LIN {X 0,Y 542.266,Z 432.631,A -85,B 0,C 180,E1 25597.331,E2 25597.331} C_VEL
LIN {X 0,Y 541.253,Z 430.993,A -85,B 0,C 180,E1 25597.163,E2 25597.163} C_VEL
LIN {X 0,Y 538.577,Z 428.153,A -85,B 0,C 180,E1 25596.746,E2 25596.746} C_VEL
LIN {X 0,Y 537.692,Z 425.915,A -85,B 0,C 180,E1 25596.518,E2 25596.518} C_VEL
LIN {X 0,Y 537.544,Z 425.203,A -85,B 0,C 180,E1 25596.133,E2 25596.133} C_VEL
LIN {X 0,Y 537.618,Z 425.265,A -85,B 0,C 180,E1 25592.894,E2 25592.894} C_VEL
LIN {X 0,Y 537.548,Z 425.178,A -85,B 0,C 180,E1 25589.656,E2 25589.656} C_VEL
LIN {X 0,Y 537.585,Z 425.269,A -85,B 0,C 180,E1 25586.275,E2 25586.275} C_VEL
LIN {X 0,Y 537.609,Z 425.252,A -85,B 0,C 180,E1 25582.979,E2 25582.979} C_VEL
LIN {X 0,Y 537.57,Z 425.245,A -85,B 0,C 180,E1 25579.674,E2 25579.674} C_VEL
LIN {X 0,Y 537.613,Z 425.237,A -85,B 0,C 180,E1 25576.322,E2 25576.322} C_VEL
LIN {X 0,Y 537.603,Z 425.259,A -85,B 0,C 180,E1 25573.006,E2 25573.006} C_VEL
LIN {X 0,Y 537.584,Z 425.263,A -85,B 0,C 180,E1 25569.637,E2 25569.637} C_VEL
LIN {X 0,Y 537.626,Z 425.237,A -85,B 0,C 180,E1 25566.3,E2 25566.3} C_VEL
LIN {X 0,Y 537.608,Z 425.241,A -85,B 0,C 180,E1 25562.878,E2 25562.878} C_VEL
LIN {X 0,Y 537.596,Z 425.261,A -85,B 0,C 180,E1 25559.467,E2 25559.467} C_VEL
LIN {X 0,Y 537.62,Z 425.243,A -85,B 0,C 180,E1 25556.054,E2 25556.054} C_VEL
LIN {X 0,Y 537.626,Z 425.232,A -85,B 0,C 180,E1 25552.627,E2 25552.627} C_VEL
LIN {X 0,Y 537.605,Z 425.254,A -85,B 0,C 180,E1 25549.173,E2 25549.173} C_VEL
LIN {X 0,Y 537.63,Z 425.26,A -85,B 0,C 180,E1 25545.679,E2 25545.679} C_VEL
LIN {X 0,Y 537.614,Z 425.246,A -85,B 0,C 180,E1 25542.224,E2 25542.224} C_VEL
LIN {X 0,Y 537.613,Z 425.226,A -85,B 0,C 180,E1 25538.85,E2 25538.85} C_VEL
LIN {X 0,Y 537.626,Z 425.262,A -85,B 0,C 180,E1 25535.38,E2 25535.38} C_VEL
LIN {X 0,Y 537.604,Z 425.242,A -85,B 0,C 180,E1 25531.93,E2 25531.93} C_VEL
LIN {X 0,Y 537.621,Z 425.229,A -85,B 0,C 180,E1 25528.613,E2 25528.613} C_VEL
LIN {X 0,Y 537.621,Z 425.237,A -85,B 0,C 180,E1 25525.182,E2 25525.182} C_VEL
LIN {X 0,Y 537.647,Z 425.416,A -85,B 0,C 180,E1 25522.998,E2 25522.998} C_VEL
LIN {X 0,Y 539.164,Z 429.093,A -85,B 0,C 180,E1 25522.266,E2 25522.266} C_VEL
LIN {X 0,Y 543.606,Z 438.861,A -85,B 0,C 180,E1 25520.474,E2 25520.474} C_VEL
LIN {X 0,Y 547.01,Z 446.029,A -85,B 0,C 180,E1 25519.264,E2 25519.264} C_VEL
LIN {X 0,Y 560.162,Z 465.654,A -85,B 0,C 180,E1 25517.289,E2 25517.289} C_VEL
LIN {X 0,Y 573.666,Z 487.219,A -85,B 0,C 180,E1 25515.413,E2 25515.413} C_VEL
LIN {X 0,Y 582.89,Z 503.607,A -85,B 0,C 180,E1 25514.188,E2 25514.188} C_VEL
LIN {X 0,Y 576.127,Z 736.515,A -85,B 0,C 180,E1 25510.926,E2 25510.926} C_VEL
LIN {X 0,Y 573.148,Z 839.663,A -85,B 0,C 180,E1 25509.472,E2 25509.472} C_VEL
LIN {X 0,Y 571.458,Z 865.731,A -85,B 0,C 180,E1 25508.946,E2 25508.946} C_VEL
LIN {X 0,Y 569.58,Z 887.597,A -85,B 0,C 180,E1 25508.349,E2 25508.349} C_VEL
LIN {X 0,Y 567.024,Z 912.5,A -85,B 0,C 180,E1 25507.472,E2 25507.472} C_VEL
LIN {X 0,Y 564.59,Z 933.033,A -85,B 0,C 180,E1 25506.58,E2 25506.58} C_VEL
LIN {X 0,Y 561.628,Z 955.658,A -85,B 0,C 180,E1 25505.413,E2 25505.413} C_VEL
LIN {X 0,Y 558.746,Z 975.609,A -85,B 0,C 180,E1 25504.188,E2 25504.188} C_VEL
LIN {X 0,Y 555.88,Z 994.545,A -85,B 0,C 180,E1 25502.858,E2 25502.858} C_VEL
LIN {X 0,Y 552.579,Z 1015.247,A -85,B 0,C 180,E1 25501.166,E2 25501.166} C_VEL
LIN {X 0,Y 549.796,Z 1032.714,A -85,B 0,C 180,E1 25499.529,E2 25499.529} C_VEL
LIN {X 0,Y 546.718,Z 1052.022,A -85,B 0,C 180,E1 25497.444,E2 25497.444} C_VEL
LIN {X 0,Y 544.377,Z 1067.179,A -85,B 0,C 180,E1 25495.572,E2 25495.572} C_VEL
LIN {X 0,Y 541.987,Z 1083.549,A -85,B 0,C 180,E1 25493.254,E2 25493.254} C_VEL
LIN {X 0,Y 540.268,Z 1096.427,A -85,B 0,C 180,E1 25491.155,E2 25491.155} C_VEL
LIN {X 0,Y 538.657,Z 1109.908,A -85,B 0,C 180,E1 25488.619,E2 25488.619} C_VEL
LIN {X 0,Y 537.638,Z 1119.894,A -85,B 0,C 180,E1 25486.421,E2 25486.421} C_VEL
LIN {X 0,Y 536.832,Z 1129.669,A -85,B 0,C 180,E1 25483.903,E2 25483.903} C_VEL
LIN {X 0,Y 536.342,Z 1137.217,A -85,B 0,C 180,E1 25481.506,E2 25481.506} C_VEL
LIN {X 0,Y 536.089,Z 1143.09,A -85,B 0,C 180,E1 25479.23,E2 25479.23} C_VEL
LIN {X 0,Y 535.96,Z 1148.292,A -85,B 0,C 180,E1 25476.535,E2 25476.535} C_VEL
LIN {X 0,Y 535.933,Z 1151.266,A -85,B 0,C 180,E1 25474.28,E2 25474.28} C_VEL
LIN {X 0,Y 535.914,Z 1153.221,A -85,B 0,C 180,E1 25471.711,E2 25471.711} C_VEL
LIN {X 0,Y 535.9,Z 1153.457,A -85,B 0,C 180,E1 25469.359,E2 25469.359} C_VEL
LIN {X 0,Y 535.9,Z 1152.559,A -85,B 0,C 180,E1 25467.219,E2 25467.219} C_VEL
LIN {X 0,Y 535.912,Z 1150.339,A -85,B 0,C 180,E1 25464.862,E2 25464.862} C_VEL
LIN {X 0,Y 535.975,Z 1146.441,A -85,B 0,C 180,E1 25462.389,E2 25462.389} C_VEL
LIN {X 0,Y 536.155,Z 1141.549,A -85,B 0,C 180,E1 25460.121,E2 25460.121} C_VEL
LIN {X 0,Y 536.518,Z 1134.571,A -85,B 0,C 180,E1 25457.572,E2 25457.572} C_VEL
LIN {X 0,Y 537.116,Z 1126.055,A -85,B 0,C 180,E1 25455.114,E2 25455.114} C_VEL
LIN {X 0,Y 538.018,Z 1116.198,A -85,B 0,C 180,E1 25452.701,E2 25452.701} C_VEL
LIN {X 0,Y 539.299,Z 1104.351,A -85,B 0,C 180,E1 25450.279,E2 25450.279} C_VEL
LIN {X 0,Y 540.858,Z 1091.93,A -85,B 0,C 180,E1 25448.072,E2 25448.072} C_VEL
LIN {X 0,Y 542.939,Z 1076.73,A -85,B 0,C 180,E1 25445.752,E2 25445.752} C_VEL
LIN {X 0,Y 545,Z 1062.711,A -85,B 0,C 180,E1 25443.876,E2 25443.876} C_VEL
LIN {X 0,Y 547.829,Z 1044.176,A -85,B 0,C 180,E1 25441.713,E2 25441.713} C_VEL
LIN {X 0,Y 550.405,Z 1027.597,A -85,B 0,C 180,E1 25440.028,E2 25440.028} C_VEL
LIN {X 0,Y 553.667,Z 1006.611,A -85,B 0,C 180,E1 25438.174,E2 25438.174} C_VEL
LIN {X 0,Y 556.354,Z 988.668,A -85,B 0,C 180,E1 25436.801,E2 25436.801} C_VEL
LIN {X 0,Y 559.46,Z 967.1,A -85,B 0,C 180,E1 25435.365,E2 25435.365} C_VEL
LIN {X 0,Y 562.201,Z 946.182,A -85,B 0,C 180,E1 25434.187,E2 25434.187} C_VEL
LIN {X 0,Y 564.963,Z 924.058,A -85,B 0,C 180,E1 25433.127,E2 25433.127} C_VEL
LIN {X 0,Y 567.281,Z 901.886,A -85,B 0,C 180,E1 25432.261,E2 25432.261} C_VEL
LIN {X 0,Y 569.212,Z 881.106,A -85,B 0,C 180,E1 25431.595,E2 25431.595} C_VEL
LIN {X 0,Y 571.144,Z 855.513,A -85,B 0,C 180,E1 25430.967,E2 25430.967} C_VEL
LIN {X 0,Y 572.245,Z 833.472,A -85,B 0,C 180,E1 25430.575,E2 25430.575} C_VEL
LIN {X 0,Y 578.309,Z 600.743,A -85,B 0,C 180,E1 25427.358,E2 25427.358} C_VEL
LIN {X 0,Y 580.866,Z 502.463,A -85,B 0,C 180,E1 25425.981,E2 25425.981} C_VEL
LIN {X 0,Y 566.803,Z 478.221,A -85,B 0,C 180,E1 25424.243,E2 25424.243} C_VEL
LIN {X 0,Y 553.848,Z 457.367,A -85,B 0,C 180,E1 25422.54,E2 25422.54} C_VEL
LIN {X 0,Y 546.451,Z 445.944,A -85,B 0,C 180,E1 25421.482,E2 25421.482} C_VEL
LIN {X 0,Y 540.732,Z 432.695,A -85,B 0,C 180,E1 25419.365,E2 25419.365} C_VEL
LIN {X 0,Y 537.629,Z 425.514,A -85,B 0,C 180,E1 25418.121,E2 25418.121} C_VEL
LIN {X 0,Y 537.624,Z 425.259,A -85,B 0,C 180,E1 25415.208,E2 25415.208} C_VEL
LIN {X 0,Y 537.61,Z 425.251,A -85,B 0,C 180,E1 25411.759,E2 25411.759} C_VEL
LIN {X 0,Y 537.608,Z 425.234,A -85,B 0,C 180,E1 25408.312,E2 25408.312} C_VEL
LIN {X 0,Y 537.616,Z 425.237,A -85,B 0,C 180,E1 25404.973,E2 25404.973} C_VEL
LIN {X 0,Y 537.624,Z 425.265,A -85,B 0,C 180,E1 25401.493,E2 25401.493} C_VEL
LIN {X 0,Y 537.613,Z 425.246,A -85,B 0,C 180,E1 25397.983,E2 25397.983} C_VEL
LIN {X 0,Y 537.609,Z 425.234,A -85,B 0,C 180,E1 25394.652,E2 25394.652} C_VEL
LIN {X 0,Y 537.615,Z 425.263,A -85,B 0,C 180,E1 25391.153,E2 25391.153} C_VEL
LIN {X 0,Y 537.618,Z 425.237,A -85,B 0,C 180,E1 25387.696,E2 25387.696} C_VEL
LIN {X 0,Y 537.606,Z 425.246,A -85,B 0,C 180,E1 25384.373,E2 25384.373} C_VEL
LIN {X 0,Y 537.6,Z 425.265,A -85,B 0,C 180,E1 25380.853,E2 25380.853} C_VEL
LIN {X 0,Y 537.62,Z 425.228,A -85,B 0,C 180,E1 25377.548,E2 25377.548} C_VEL
LIN {X 0,Y 537.597,Z 425.262,A -85,B 0,C 180,E1 25374.236,E2 25374.236} C_VEL
LIN {X 0,Y 537.591,Z 425.241,A -85,B 0,C 180,E1 25370.796,E2 25370.796} C_VEL
LIN {X 0,Y 537.627,Z 425.238,A -85,B 0,C 180,E1 25367.432,E2 25367.432} C_VEL
LIN {X 0,Y 537.582,Z 425.264,A -85,B 0,C 180,E1 25364.132,E2 25364.132} C_VEL
LIN {X 0,Y 537.58,Z 425.237,A -85,B 0,C 180,E1 25360.666,E2 25360.666} C_VEL
LIN {X 0,Y 537.635,Z 425.243,A -85,B 0,C 180,E1 25357.358,E2 25357.358} C_VEL
LIN {X 0,Y 537.568,Z 425.266,A -85,B 0,C 180,E1 25354.08,E2 25354.08} C_VEL
LIN {X 0,Y 537.583,Z 425.243,A -85,B 0,C 180,E1 25350.714,E2 25350.714} C_VEL
LIN {X 0,Y 537.577,Z 425.245,A -85,B 0,C 180,E1 25347.61,E2 25347.61} C_VEL
LIN {X 0,Y 537.553,Z 425.26,A -85,B 0,C 180,E1 25344.263,E2 25344.263} C_VEL
LIN {X 0,Y 537.625,Z 425.26,A -85,B 0,C 180,E1 25341.024,E2 25341.024} C_VEL
LIN {X 0,Y 537.534,Z 425.176,A -85,B 0,C 180,E1 25337.76,E2 25337.76} C_VEL
LIN {X 0,Y 537.597,Z 425.501,A -85,B 0,C 180,E1 25336.5,E2 25336.5} C_VEL
LIN {X 0,Y 538.028,Z 427.128,A -85,B 0,C 180,E1 25336.29,E2 25336.29} C_VEL
LIN {X 0,Y 540.035,Z 430.094,A -85,B 0,C 180,E1 25335.989,E2 25335.989} C_VEL
LIN {X 0,Y 541.571,Z 431.696,A -85,B 0,C 180,E1 25335.778,E2 25335.778} C_VEL
LIN {X 0,Y 544.264,Z 435.602,A -85,B 0,C 180,E1 25335.392,E2 25335.392} C_VEL
LIN {X 0,Y 546.005,Z 438.026,A -85,B 0,C 180,E1 25335.148,E2 25335.148} C_VEL
LIN {X 0,Y 556.165,Z 451.925,A -85,B 0,C 180,E1 25333.775,E2 25333.775} C_VEL
LIN {X 0,Y 568.902,Z 470.607,A -85,B 0,C 180,E1 25332.142,E2 25332.142} C_VEL
LIN {X 0,Y 578.998,Z 486.605,A -85,B 0,C 180,E1 25330.909,E2 25330.909} C_VEL
LIN {X 0,Y 581.084,Z 490.587,A -85,B 0,C 180,E1 25330.651,E2 25330.651} C_VEL
LIN {X 0,Y 574.372,Z 738.934,A -85,B 0,C 180,E1 25327.219,E2 25327.219} C_VEL
LIN {X 0,Y 573.077,Z 788.809,A -85,B 0,C 180,E1 25326.536,E2 25326.536} C_VEL
LIN {X 0,Y 572.103,Z 796.494,A -85,B 0,C 180,E1 25326.491,E2 25326.491} C_VEL
LIN {X 0,Y 566.562,Z 815.841,A -85,B 0,C 180,E1 25326.555,E2 25326.555} C_VEL
LIN {X 0,Y 565.37,Z 823.458,A -85,B 0,C 180,E1 25326.46,E2 25326.46} C_VEL
LIN {X 0,Y 563.471,Z 849.649,A -85,B 0,C 180,E1 25325.798,E2 25325.798} C_VEL
LIN {X 0,Y 561.563,Z 870.523,A -85,B 0,C 180,E1 25325.108,E2 25325.108} C_VEL
LIN {X 0,Y 558.954,Z 894.83,A -85,B 0,C 180,E1 25324.112,E2 25324.112} C_VEL
LIN {X 0,Y 556.401,Z 914.903,A -85,B 0,C 180,E1 25323.114,E2 25323.114} C_VEL
LIN {X 0,Y 553.426,Z 936.721,A -85,B 0,C 180,E1 25321.841,E2 25321.841} C_VEL
LIN {X 0,Y 550.342,Z 956.701,A -85,B 0,C 180,E1 25320.458,E2 25320.458} C_VEL
LIN {X 0,Y 547.295,Z 975.651,A -85,B 0,C 180,E1 25318.957,E2 25318.957} C_VEL
LIN {X 0,Y 544.056,Z 994.807,A -85,B 0,C 180,E1 25317.187,E2 25317.187} C_VEL
LIN {X 0,Y 541.331,Z 1010.879,A -85,B 0,C 180,E1 25315.491,E2 25315.491} C_VEL
LIN {X 0,Y 538.391,Z 1028.003,A -85,B 0,C 180,E1 25313.418,E2 25313.418} C_VEL
LIN {X 0,Y 536.15,Z 1041.437,A -85,B 0,C 180,E1 25311.555,E2 25311.555} C_VEL
LIN {X 0,Y 533.853,Z 1056.035,A -85,B 0,C 180,E1 25309.247,E2 25309.247} C_VEL
LIN {X 0,Y 532.096,Z 1067.944,A -85,B 0,C 180,E1 25307.047,E2 25307.047} C_VEL
LIN {X 0,Y 530.614,Z 1079.355,A -85,B 0,C 180,E1 25304.626,E2 25304.626} C_VEL
LIN {X 0,Y 529.486,Z 1089.213,A -85,B 0,C 180,E1 25302.1,E2 25302.1} C_VEL
LIN {X 0,Y 528.768,Z 1097.158,A -85,B 0,C 180,E1 25299.689,E2 25299.689} C_VEL
LIN {X 0,Y 528.286,Z 1104.028,A -85,B 0,C 180,E1 25297.067,E2 25297.067} C_VEL
LIN {X 0,Y 528.073,Z 1108.717,A -85,B 0,C 180,E1 25294.779,E2 25294.779} C_VEL
LIN {X 0,Y 527.969,Z 1112.732,A -85,B 0,C 180,E1 25292.062,E2 25292.062} C_VEL
LIN {X 0,Y 527.938,Z 1114.802,A -85,B 0,C 180,E1 25289.674,E2 25289.674} C_VEL
LIN {X 0,Y 527.922,Z 1115.688,A -85,B 0,C 180,E1 25287.177,E2 25287.177} C_VEL
LIN {X 0,Y 527.93,Z 1115.011,A -85,B 0,C 180,E1 25284.566,E2 25284.566} C_VEL
LIN {X 0,Y 527.961,Z 1113.176,A -85,B 0,C 180,E1 25282.272,E2 25282.272} C_VEL
LIN {X 0,Y 528.057,Z 1109.669,A -85,B 0,C 180,E1 25279.637,E2 25279.637} C_VEL
LIN {X 0,Y 528.264,Z 1104.62,A -85,B 0,C 180,E1 25277.094,E2 25277.094} C_VEL
LIN {X 0,Y 528.691,Z 1098.426,A -85,B 0,C 180,E1 25274.646,E2 25274.646} C_VEL
LIN {X 0,Y 529.407,Z 1090.185,A -85,B 0,C 180,E1 25272.07,E2 25272.07} C_VEL
LIN {X 0,Y 530.357,Z 1081.59,A -85,B 0,C 180,E1 25269.817,E2 25269.817} C_VEL
LIN {X 0,Y 531.952,Z 1069.284,A -85,B 0,C 180,E1 25267.102,E2 25267.102} C_VEL
LIN {X 0,Y 533.624,Z 1057.85,A -85,B 0,C 180,E1 25264.946,E2 25264.946} C_VEL
LIN {X 0,Y 536.117,Z 1042.465,A -85,B 0,C 180,E1 25262.449,E2 25262.449} C_VEL
LIN {X 0,Y 538.46,Z 1028.763,A -85,B 0,C 180,E1 25260.522,E2 25260.522} C_VEL
LIN {X 0,Y 541.631,Z 1010.837,A -85,B 0,C 180,E1 25258.326,E2 25258.326} C_VEL
LIN {X 0,Y 544.479,Z 994.653,A -85,B 0,C 180,E1 25256.605,E2 25256.605} C_VEL
LIN {X 0,Y 547.931,Z 975.025,A -85,B 0,C 180,E1 25254.784,E2 25254.784} C_VEL
LIN {X 0,Y 550.968,Z 956.873,A -85,B 0,C 180,E1 25253.335,E2 25253.335} C_VEL
LIN {X 0,Y 554.273,Z 936.366,A -85,B 0,C 180,E1 25251.905,E2 25251.905} C_VEL
LIN {X 0,Y 557.315,Z 914.937,A -85,B 0,C 180,E1 25250.648,E2 25250.648} C_VEL
LIN {X 0,Y 560.096,Z 894.066,A -85,B 0,C 180,E1 25249.606,E2 25249.606} C_VEL
LIN {X 0,Y 562.694,Z 870.908,A -85,B 0,C 180,E1 25248.655,E2 25248.655} C_VEL
LIN {X 0,Y 564.75,Z 849.402,A -85,B 0,C 180,E1 25247.939,E2 25247.939} C_VEL
LIN {X 0,Y 566.716,Z 823.568,A -85,B 0,C 180,E1 25247.286,E2 25247.286} C_VEL
LIN {X 0,Y 567.823,Z 801.817,A -85,B 0,C 180,E1 25246.888,E2 25246.888} C_VEL
LIN {X 0,Y 575.439,Z 551.354,A -85,B 0,C 180,E1 25243.354,E2 25243.354} C_VEL
LIN {X 0,Y 577.148,Z 493.917,A -85,B 0,C 180,E1 25242.527,E2 25242.527} C_VEL
LIN {X 0,Y 568.475,Z 480.151,A -85,B 0,C 180,E1 25241.369,E2 25241.369} C_VEL
LIN {X 0,Y 556.198,Z 462.48,A -85,B 0,C 180,E1 25239.657,E2 25239.657} C_VEL
LIN {X 0,Y 545.014,Z 447.399,A -85,B 0,C 180,E1 25237.989,E2 25237.989} C_VEL
LIN {X 0,Y 541.363,Z 442.627,A -85,B 0,C 180,E1 25237.419,E2 25237.419} C_VEL
LIN {X 0,Y 538.138,Z 438.133,A -85,B 0,C 180,E1 25236.898,E2 25236.898} C_VEL
LIN {X 0,Y 534.685,Z 434.016,A -85,B 0,C 180,E1 25236.34,E2 25236.34} C_VEL
LIN {X 0,Y 533.712,Z 432.247,A -85,B 0,C 180,E1 25236.167,E2 25236.167} C_VEL
LIN {X 0,Y 530.926,Z 429.69,A -85,B 0,C 180,E1 25235.72,E2 25235.72} C_VEL
LIN {X 0,Y 529.78,Z 427.076,A -85,B 0,C 180,E1 25235.455,E2 25235.455} C_VEL
LIN {X 0,Y 529.652,Z 426.247,A -85,B 0,C 180,E1 25235.155,E2 25235.155} C_VEL
LIN {X 0,Y 529.611,Z 426.213,A -85,B 0,C 180,E1 25231.913,E2 25231.913} C_VEL
LIN {X 0,Y 529.669,Z 426.168,A -85,B 0,C 180,E1 25228.62,E2 25228.62} C_VEL
LIN {X 0,Y 529.636,Z 426.248,A -85,B 0,C 180,E1 25225.376,E2 25225.376} C_VEL
LIN {X 0,Y 529.633,Z 426.257,A -85,B 0,C 180,E1 25221.95,E2 25221.95} C_VEL
LIN {X 0,Y 529.687,Z 426.245,A -85,B 0,C 180,E1 25218.604,E2 25218.604} C_VEL
LIN {X 0,Y 529.642,Z 426.23,A -85,B 0,C 180,E1 25215.269,E2 25215.269} C_VEL
LIN {X 0,Y 529.644,Z 426.229,A -85,B 0,C 180,E1 25211.764,E2 25211.764} C_VEL
LIN {X 0,Y 529.691,Z 426.243,A -85,B 0,C 180,E1 25208.358,E2 25208.358} C_VEL
LIN {X 0,Y 529.665,Z 426.247,A -85,B 0,C 180,E1 25204.982,E2 25204.982} C_VEL
LIN {X 0,Y 529.651,Z 426.223,A -85,B 0,C 180,E1 25201.515,E2 25201.515} C_VEL
LIN {X 0,Y 529.684,Z 426.227,A -85,B 0,C 180,E1 25198.161,E2 25198.161} C_VEL
LIN {X 0,Y 529.681,Z 426.249,A -85,B 0,C 180,E1 25194.693,E2 25194.693} C_VEL
LIN {X 0,Y 529.663,Z 426.236,A -85,B 0,C 180,E1 25191.314,E2 25191.314} C_VEL
LIN {X 0,Y 529.679,Z 426.221,A -85,B 0,C 180,E1 25187.905,E2 25187.905} C_VEL
LIN {X 0,Y 529.683,Z 426.238,A -85,B 0,C 180,E1 25184.451,E2 25184.451} C_VEL
LIN {X 0,Y 529.677,Z 426.254,A -85,B 0,C 180,E1 25180.939,E2 25180.939} C_VEL
LIN {X 0,Y 529.689,Z 426.215,A -85,B 0,C 180,E1 25177.468,E2 25177.468} C_VEL
LIN {X 0,Y 529.665,Z 426.22,A -85,B 0,C 180,E1 25174.026,E2 25174.026} C_VEL
LIN {X 0,Y 529.69,Z 426.25,A -85,B 0,C 180,E1 25170.607,E2 25170.607} C_VEL
LIN {X 0,Y 529.686,Z 426.24,A -85,B 0,C 180,E1 25167.067,E2 25167.067} C_VEL
LIN {X 0,Y 529.686,Z 426.433,A -85,B 0,C 180,E1 25164.012,E2 25164.012} C_VEL
LIN {X 0,Y 531.268,Z 430.136,A -85,B 0,C 180,E1 25163.237,E2 25163.237} C_VEL
LIN {X 0,Y 537.41,Z 443.418,A -85,B 0,C 180,E1 25160.715,E2 25160.715} C_VEL
LIN {X 0,Y 538.748,Z 446.108,A -85,B 0,C 180,E1 25160.324,E2 25160.324} C_VEL
LIN {X 0,Y 547.604,Z 458.825,A -85,B 0,C 180,E1 25158.92,E2 25158.92} C_VEL
LIN {X 0,Y 559.849,Z 477.44,A -85,B 0,C 180,E1 25157.102,E2 25157.102} C_VEL
LIN {X 0,Y 570.86,Z 495.65,A -85,B 0,C 180,E1 25155.558,E2 25155.558} C_VEL
LIN {X 0,Y 577.15,Z 506.92,A -85,B 0,C 180,E1 25154.706,E2 25154.706} C_VEL
LIN {X 0,Y 570.13,Z 737.84,A -85,B 0,C 180,E1 25151.445,E2 25151.445} C_VEL
LIN {X 0,Y 567.06,Z 839.446,A -85,B 0,C 180,E1 25149.999,E2 25149.999} C_VEL
LIN {X 0,Y 565.316,Z 865.417,A -85,B 0,C 180,E1 25149.472,E2 25149.472} C_VEL
LIN {X 0,Y 563.366,Z 887.233,A -85,B 0,C 180,E1 25148.873,E2 25148.873} C_VEL
LIN {X 0,Y 560.635,Z 912.63,A -85,B 0,C 180,E1 25147.972,E2 25147.972} C_VEL
LIN {X 0,Y 558.106,Z 933.07,A -85,B 0,C 180,E1 25147.076,E2 25147.076} C_VEL
LIN {X 0,Y 554.879,Z 956.488,A -85,B 0,C 180,E1 25145.849,E2 25145.849} C_VEL
LIN {X 0,Y 552.005,Z 975.542,A -85,B 0,C 180,E1 25144.665,E2 25144.665} C_VEL
LIN {X 0,Y 548.867,Z 995.372,A -85,B 0,C 180,E1 25143.254,E2 25143.254} C_VEL
LIN {X 0,Y 545.439,Z 1015.723,A -85,B 0,C 180,E1 25141.559,E2 25141.559} C_VEL
LIN {X 0,Y 542.351,Z 1034.232,A -85,B 0,C 180,E1 25139.792,E2 25139.792} C_VEL
LIN {X 0,Y 539.365,Z 1051.939,A -85,B 0,C 180,E1 25137.837,E2 25137.837} C_VEL
LIN {X 0,Y 536.902,Z 1066.971,A -85,B 0,C 180,E1 25135.954,E2 25135.954} C_VEL
LIN {X 0,Y 534.381,Z 1083.314,A -85,B 0,C 180,E1 25133.605,E2 25133.605} C_VEL
LIN {X 0,Y 532.543,Z 1096.174,A -85,B 0,C 180,E1 25131.477,E2 25131.477} C_VEL
LIN {X 0,Y 530.83,Z 1109.631,A -85,B 0,C 180,E1 25128.904,E2 25128.904} C_VEL
LIN {X 0,Y 529.75,Z 1119.601,A -85,B 0,C 180,E1 25126.672,E2 25126.672} C_VEL
LIN {X 0,Y 528.885,Z 1129.419,A -85,B 0,C 180,E1 25124.102,E2 25124.102} C_VEL
LIN {X 0,Y 528.372,Z 1136.924,A -85,B 0,C 180,E1 25121.682,E2 25121.682} C_VEL
LIN {X 0,Y 528.106,Z 1142.8,A -85,B 0,C 180,E1 25119.371,E2 25119.371} C_VEL
LIN {X 0,Y 527.965,Z 1148.004,A -85,B 0,C 180,E1 25116.634,E2 25116.634} C_VEL
LIN {X 0,Y 527.935,Z 1150.979,A -85,B 0,C 180,E1 25114.345,E2 25114.345} C_VEL
LIN {X 0,Y 527.922,Z 1152.896,A -85,B 0,C 180,E1 25111.845,E2 25111.845} C_VEL
LIN {X 0,Y 527.905,Z 1153.172,A -85,B 0,C 180,E1 25109.349,E2 25109.349} C_VEL
LIN {X 0,Y 527.903,Z 1152.275,A -85,B 0,C 180,E1 25107.177,E2 25107.177} C_VEL
LIN {X 0,Y 527.914,Z 1150.054,A -85,B 0,C 180,E1 25104.784,E2 25104.784} C_VEL
LIN {X 0,Y 527.992,Z 1145.945,A -85,B 0,C 180,E1 25102.163,E2 25102.163} C_VEL
LIN {X 0,Y 528.175,Z 1141.033,A -85,B 0,C 180,E1 25099.873,E2 25099.873} C_VEL
LIN {X 0,Y 528.588,Z 1133.736,A -85,B 0,C 180,E1 25097.213,E2 25097.213} C_VEL
LIN {X 0,Y 529.194,Z 1125.766,A -85,B 0,C 180,E1 25094.886,E2 25094.886} C_VEL
LIN {X 0,Y 530.1,Z 1116.369,A -85,B 0,C 180,E1 25092.548,E2 25092.548} C_VEL
LIN {X 0,Y 531.442,Z 1104.615,A -85,B 0,C 180,E1 25090.09,E2 25090.09} C_VEL
LIN {X 0,Y 532.979,Z 1092.886,A -85,B 0,C 180,E1 25087.963,E2 25087.963} C_VEL
LIN {X 0,Y 535.249,Z 1077.15,A -85,B 0,C 180,E1 25085.499,E2 25085.499} C_VEL
LIN {X 0,Y 537.402,Z 1063.189,A -85,B 0,C 180,E1 25083.597,E2 25083.597} C_VEL
LIN {X 0,Y 540.332,Z 1044.933,A -85,B 0,C 180,E1 25081.422,E2 25081.422} C_VEL
LIN {X 0,Y 543.038,Z 1028.296,A -85,B 0,C 180,E1 25079.701,E2 25079.701} C_VEL
LIN {X 0,Y 546.23,Z 1008.857,A -85,B 0,C 180,E1 25077.937,E2 25077.937} C_VEL
LIN {X 0,Y 549.187,Z 989.911,A -85,B 0,C 180,E1 25076.456,E2 25076.456} C_VEL
LIN {X 0,Y 552.38,Z 968.924,A -85,B 0,C 180,E1 25075.023,E2 25075.023} C_VEL
LIN {X 0,Y 555.395,Z 946.898,A -85,B 0,C 180,E1 25073.76,E2 25073.76} C_VEL
LIN {X 0,Y 558.219,Z 925.153,A -85,B 0,C 180,E1 25072.702,E2 25072.702} C_VEL
LIN {X 0,Y 560.785,Z 901.912,A -85,B 0,C 180,E1 25071.778,E2 25071.778} C_VEL
LIN {X 0,Y 562.747,Z 881.616,A -85,B 0,C 180,E1 25071.121,E2 25071.121} C_VEL
LIN {X 0,Y 564.78,Z 856,A -85,B 0,C 180,E1 25070.481,E2 25070.481} C_VEL
LIN {X 0,Y 565.948,Z 833.625,A -85,B 0,C 180,E1 25070.077,E2 25070.077} C_VEL
LIN {X 0,Y 572.285,Z 601.478,A -85,B 0,C 180,E1 25066.839,E2 25066.839} C_VEL
LIN {X 0,Y 574.899,Z 505.729,A -85,B 0,C 180,E1 25065.487,E2 25065.487} C_VEL
LIN {X 0,Y 560.515,Z 480.862,A -85,B 0,C 180,E1 25063.659,E2 25063.659} C_VEL
LIN {X 0,Y 548.607,Z 461.767,A -85,B 0,C 180,E1 25062.052,E2 25062.052} C_VEL
LIN {X 0,Y 538.073,Z 445.468,A -85,B 0,C 180,E1 25060.502,E2 25060.502} C_VEL
LIN {X 0,Y 532.475,Z 433.182,A -85,B 0,C 180,E1 25058.43,E2 25058.43} C_VEL
LIN {X 0,Y 529.704,Z 426.379,A -85,B 0,C 180,E1 25057.205,E2 25057.205} C_VEL
LIN {X 0,Y 529.672,Z 426.232,A -85,B 0,C 180,E1 25053.711,E2 25053.711} C_VEL
LIN {X 0,Y 529.664,Z 426.246,A -85,B 0,C 180,E1 25050.268,E2 25050.268} C_VEL
LIN {X 0,Y 529.682,Z 426.248,A -85,B 0,C 180,E1 25046.94,E2 25046.94} C_VEL
LIN {X 0,Y 529.681,Z 426.22,A -85,B 0,C 180,E1 25043.446,E2 25043.446} C_VEL
LIN {X 0,Y 529.673,Z 426.231,A -85,B 0,C 180,E1 25040.095,E2 25040.095} C_VEL
LIN {X 0,Y 529.677,Z 426.251,A -85,B 0,C 180,E1 25036.675,E2 25036.675} C_VEL
LIN {X 0,Y 529.678,Z 426.224,A -85,B 0,C 180,E1 25033.204,E2 25033.204} C_VEL
LIN {X 0,Y 529.677,Z 426.228,A -85,B 0,C 180,E1 25029.782,E2 25029.782} C_VEL
LIN {X 0,Y 529.673,Z 426.25,A -85,B 0,C 180,E1 25026.395,E2 25026.395} C_VEL
LIN {X 0,Y 529.66,Z 426.219,A -85,B 0,C 180,E1 25022.922,E2 25022.922} C_VEL
LIN {X 0,Y 529.686,Z 426.246,A -85,B 0,C 180,E1 25019.567,E2 25019.567} C_VEL
LIN {X 0,Y 529.668,Z 426.236,A -85,B 0,C 180,E1 25016.103,E2 25016.103} C_VEL
LIN {X 0,Y 529.649,Z 426.226,A -85,B 0,C 180,E1 25012.733,E2 25012.733} C_VEL
LIN {X 0,Y 529.686,Z 426.25,A -85,B 0,C 180,E1 25009.339,E2 25009.339} C_VEL
LIN {X 0,Y 529.65,Z 426.219,A -85,B 0,C 180,E1 25006.013,E2 25006.013} C_VEL
LIN {X 0,Y 529.64,Z 426.244,A -85,B 0,C 180,E1 25002.532,E2 25002.532} C_VEL
LIN {X 0,Y 529.683,Z 426.244,A -85,B 0,C 180,E1 24999.135,E2 24999.135} C_VEL
LIN {X 0,Y 529.635,Z 426.221,A -85,B 0,C 180,E1 24995.934,E2 24995.934} C_VEL
LIN {X 0,Y 529.628,Z 426.24,A -85,B 0,C 180,E1 24992.449,E2 24992.449} C_VEL
LIN {X 0,Y 529.69,Z 426.252,A -85,B 0,C 180,E1 24989.194,E2 24989.194} C_VEL
LIN {X 0,Y 529.618,Z 426.247,A -85,B 0,C 180,E1 24985.894,E2 24985.894} C_VEL
LIN {X 0,Y 529.62,Z 426.24,A -85,B 0,C 180,E1 24982.424,E2 24982.424} C_VEL
LIN {X 0,Y 529.619,Z 426.187,A -85,B 0,C 180,E1 24979.499,E2 24979.499} C_VEL
LIN {X 0,Y 529.651,Z 426.441,A -85,B 0,C 180,E1 24977.48,E2 24977.48} C_VEL
LIN {X 0,Y 530.079,Z 427.976,A -85,B 0,C 180,E1 24977.247,E2 24977.247} C_VEL
LIN {X 0,Y 532.154,Z 431.046,A -85,B 0,C 180,E1 24976.921,E2 24976.921} C_VEL
LIN {X 0,Y 533.66,Z 432.622,A -85,B 0,C 180,E1 24976.705,E2 24976.705} C_VEL
LIN {X 0,Y 536.294,Z 436.535,A -85,B 0,C 180,E1 24976.308,E2 24976.308} C_VEL
LIN {X 0,Y 537.945,Z 438.597,A -85,B 0,C 180,E1 24976.071,E2 24976.071} C_VEL
LIN {X 0,Y 551.932,Z 457.837,A -85,B 0,C 180,E1 24974.122,E2 24974.122} C_VEL
LIN {X 0,Y 564.97,Z 477.126,A -85,B 0,C 180,E1 24972.419,E2 24972.419} C_VEL
LIN {X 0,Y 574.835,Z 493.001,A -85,B 0,C 180,E1 24971.19,E2 24971.19} C_VEL
LIN {X 0,Y 575.112,Z 494.334,A -85,B 0,C 180,E1 24971.142,E2 24971.142} C_VEL
LIN {X 0,Y 568.126,Z 741.643,A -85,B 0,C 180,E1 24967.695,E2 24967.695} C_VEL
LIN {X 0,Y 566.121,Z 809.613,A -85,B 0,C 180,E1 24966.729,E2 24966.729} C_VEL
LIN {X 0,Y 565.37,Z 823.458,A -85,B 0,C 180,E1 24966.46,E2 24966.46} C_VEL
LIN {X 0,Y 563.494,Z 833.207,A -85,B 0,C 180,E1 24966.343,E2 24966.343} C_VEL
LIN {X 0,Y 558.145,Z 849.089,A -85,B 0,C 180,E1 24966.253,E2 24966.253} C_VEL
LIN {X 0,Y 556.611,Z 856.534,A -85,B 0,C 180,E1 24966.097,E2 24966.097} C_VEL
LIN {X 0,Y 556.509,Z 857.594,A -85,B 0,C 180,E1 24966.065,E2 24966.065} C_VEL
LIN {X 0,Y 554.074,Z 881.465,A -85,B 0,C 180,E1 24965.192,E2 24965.192} C_VEL
LIN {X 0,Y 551.685,Z 901.28,A -85,B 0,C 180,E1 24964.31,E2 24964.31} C_VEL
LIN {X 0,Y 548.708,Z 923.455,A -85,B 0,C 180,E1 24963.14,E2 24963.14} C_VEL
LIN {X 0,Y 545.615,Z 943.821,A -85,B 0,C 180,E1 24961.856,E2 24961.856} C_VEL
LIN {X 0,Y 542.281,Z 964.56,A -85,B 0,C 180,E1 24960.346,E2 24960.346} C_VEL
LIN {X 0,Y 538.995,Z 983.557,A -85,B 0,C 180,E1 24958.716,E2 24958.716} C_VEL
LIN {X 0,Y 535.861,Z 1001.494,A -85,B 0,C 180,E1 24956.964,E2 24956.964} C_VEL
LIN {X 0,Y 532.679,Z 1018.929,A -85,B 0,C 180,E1 24954.983,E2 24954.983} C_VEL
LIN {X 0,Y 530.113,Z 1033.496,A -85,B 0,C 180,E1 24953.099,E2 24953.099} C_VEL
LIN {X 0,Y 527.412,Z 1049.151,A -85,B 0,C 180,E1 24950.764,E2 24950.764} C_VEL
LIN {X 0,Y 525.509,Z 1060.858,A -85,B 0,C 180,E1 24948.757,E2 24948.757} C_VEL
LIN {X 0,Y 523.584,Z 1073.823,A -85,B 0,C 180,E1 24946.19,E2 24946.19} C_VEL
LIN {X 0,Y 522.325,Z 1083.463,A -85,B 0,C 180,E1 24943.937,E2 24943.937} C_VEL
LIN {X 0,Y 521.311,Z 1092.783,A -85,B 0,C 180,E1 24941.394,E2 24941.394} C_VEL
LIN {X 0,Y 520.621,Z 1100.307,A -85,B 0,C 180,E1 24938.838,E2 24938.838} C_VEL
LIN {X 0,Y 520.239,Z 1106.148,A -85,B 0,C 180,E1 24936.4,E2 24936.4} C_VEL
LIN {X 0,Y 520.009,Z 1110.997,A -85,B 0,C 180,E1 24933.664,E2 24933.664} C_VEL
LIN {X 0,Y 519.948,Z 1113.727,A -85,B 0,C 180,E1 24931.433,E2 24931.433} C_VEL
LIN {X 0,Y 519.918,Z 1115.583,A -85,B 0,C 180,E1 24928.898,E2 24928.898} C_VEL
LIN {X 0,Y 519.92,Z 1115.877,A -85,B 0,C 180,E1 24926.251,E2 24926.251} C_VEL
LIN {X 0,Y 519.947,Z 1114.936,A -85,B 0,C 180,E1 24923.929,E2 24923.929} C_VEL
LIN {X 0,Y 519.999,Z 1112.289,A -85,B 0,C 180,E1 24921.151,E2 24921.151} C_VEL
LIN {X 0,Y 520.126,Z 1108.446,A -85,B 0,C 180,E1 24918.692,E2 24918.692} C_VEL
LIN {X 0,Y 520.436,Z 1103.047,A -85,B 0,C 180,E1 24916.104,E2 24916.104} C_VEL
LIN {X 0,Y 520.997,Z 1095.872,A -85,B 0,C 180,E1 24913.498,E2 24913.498} C_VEL
LIN {X 0,Y 521.778,Z 1088.256,A -85,B 0,C 180,E1 24911.203,E2 24911.203} C_VEL
LIN {X 0,Y 523.145,Z 1077.354,A -85,B 0,C 180,E1 24908.471,E2 24908.471} C_VEL
LIN {X 0,Y 524.62,Z 1067.1,A -85,B 0,C 180,E1 24906.287,E2 24906.287} C_VEL
LIN {X 0,Y 526.881,Z 1053.31,A -85,B 0,C 180,E1 24903.757,E2 24903.757} C_VEL
LIN {X 0,Y 529.139,Z 1040.206,A -85,B 0,C 180,E1 24901.686,E2 24901.686} C_VEL
LIN {X 0,Y 532.118,Z 1024.029,A -85,B 0,C 180,E1 24899.45,E2 24899.45} C_VEL
LIN {X 0,Y 535.109,Z 1007.712,A -85,B 0,C 180,E1 24897.506,E2 24897.506} C_VEL
LIN {X 0,Y 538.498,Z 989.81,A -85,B 0,C 180,E1 24895.634,E2 24895.634} C_VEL
LIN {X 0,Y 541.882,Z 970.902,A -85,B 0,C 180,E1 24893.94,E2 24893.94} C_VEL
LIN {X 0,Y 545.258,Z 951.625,A -85,B 0,C 180,E1 24892.429,E2 24892.429} C_VEL
LIN {X 0,Y 548.595,Z 930.715,A -85,B 0,C 180,E1 24891.037,E2 24891.037} C_VEL
LIN {X 0,Y 551.606,Z 910.443,A -85,B 0,C 180,E1 24889.878,E2 24889.878} C_VEL
LIN {X 0,Y 554.66,Z 887.442,A -85,B 0,C 180,E1 24888.784,E2 24888.784} C_VEL
LIN {X 0,Y 556.918,Z 867.452,A -85,B 0,C 180,E1 24887.995,E2 24887.995} C_VEL
LIN {X 0,Y 559.256,Z 843.26,A -85,B 0,C 180,E1 24887.225,E2 24887.225} C_VEL
LIN {X 0,Y 560.842,Z 821.279,A -85,B 0,C 180,E1 24886.698,E2 24886.698} C_VEL
LIN {X 0,Y 562.007,Z 798.053,A -85,B 0,C 180,E1 24886.286,E2 24886.286} C_VEL
LIN {X 0,Y 569.944,Z 546.909,A -85,B 0,C 180,E1 24882.72,E2 24882.72} C_VEL
LIN {X 0,Y 571.44,Z 497.364,A -85,B 0,C 180,E1 24881.996,E2 24881.996} C_VEL
LIN {X 0,Y 563.163,Z 484.358,A -85,B 0,C 180,E1 24880.865,E2 24880.865} C_VEL
LIN {X 0,Y 551.891,Z 468.093,A -85,B 0,C 180,E1 24879.254,E2 24879.254} C_VEL
LIN {X 0,Y 541.102,Z 453.443,A -85,B 0,C 180,E1 24877.609,E2 24877.609} C_VEL
LIN {X 0,Y 537.066,Z 448.255,A -85,B 0,C 180,E1 24876.967,E2 24876.967} C_VEL
LIN {X 0,Y 533.515,Z 443.51,A -85,B 0,C 180,E1 24876.383,E2 24876.383} C_VEL
LIN {X 0,Y 529.862,Z 438.692,A -85,B 0,C 180,E1 24875.766,E2 24875.766} C_VEL
LIN {X 0,Y 526.909,Z 435.251,A -85,B 0,C 180,E1 24875.265,E2 24875.265} C_VEL
LIN {X 0,Y 525.771,Z 433.204,A -85,B 0,C 180,E1 24875.053,E2 24875.053} C_VEL
LIN {X 0,Y 522.929,Z 430.546,A -85,B 0,C 180,E1 24874.57,E2 24874.57} C_VEL
LIN {X 0,Y 521.822,Z 427.993,A -85,B 0,C 180,E1 24874.288,E2 24874.288} C_VEL
LIN {X 0,Y 521.673,Z 427.238,A -85,B 0,C 180,E1 24873.901,E2 24873.901} C_VEL
LIN {X 0,Y 521.72,Z 427.152,A -85,B 0,C 180,E1 24870.624,E2 24870.624} C_VEL
LIN {X 0,Y 521.69,Z 427.199,A -85,B 0,C 180,E1 24867.387,E2 24867.387} C_VEL
LIN {X 0,Y 521.689,Z 427.222,A -85,B 0,C 180,E1 24863.902,E2 24863.902} C_VEL
LIN {X 0,Y 521.748,Z 427.215,A -85,B 0,C 180,E1 24860.648,E2 24860.648} C_VEL
LIN {X 0,Y 521.706,Z 427.235,A -85,B 0,C 180,E1 24857.282,E2 24857.282} C_VEL
LIN {X 0,Y 521.705,Z 427.244,A -85,B 0,C 180,E1 24853.748,E2 24853.748} C_VEL
LIN {X 0,Y 521.746,Z 427.221,A -85,B 0,C 180,E1 24850.378,E2 24850.378} C_VEL
LIN {X 0,Y 521.727,Z 427.213,A -85,B 0,C 180,E1 24846.935,E2 24846.935} C_VEL
LIN {X 0,Y 521.713,Z 427.234,A -85,B 0,C 180,E1 24843.516,E2 24843.516} C_VEL
LIN {X 0,Y 521.75,Z 427.235,A -85,B 0,C 180,E1 24840,E2 24840} C_VEL
LIN {X 0,Y 521.74,Z 427.211,A -85,B 0,C 180,E1 24836.484,E2 24836.484} C_VEL
LIN {X 0,Y 521.724,Z 427.214,A -85,B 0,C 180,E1 24833.065,E2 24833.065} C_VEL
LIN {X 0,Y 521.735,Z 427.238,A -85,B 0,C 180,E1 24829.51,E2 24829.51} C_VEL
LIN {X 0,Y 521.738,Z 427.237,A -85,B 0,C 180,E1 24826.026,E2 24826.026} C_VEL
LIN {X 0,Y 521.739,Z 427.216,A -85,B 0,C 180,E1 24822.604,E2 24822.604} C_VEL
LIN {X 0,Y 521.734,Z 427.204,A -85,B 0,C 180,E1 24819.117,E2 24819.117} C_VEL
LIN {X 0,Y 521.735,Z 427.242,A -85,B 0,C 180,E1 24815.787,E2 24815.787} C_VEL
LIN {X 0,Y 521.731,Z 427.209,A -85,B 0,C 180,E1 24812.244,E2 24812.244} C_VEL
LIN {X 0,Y 521.741,Z 427.204,A -85,B 0,C 180,E1 24808.839,E2 24808.839} C_VEL
LIN {X 0,Y 521.731,Z 427.217,A -85,B 0,C 180,E1 24805.439,E2 24805.439} C_VEL
LIN {X 0,Y 521.823,Z 427.717,A -85,B 0,C 180,E1 24804.996,E2 24804.996} C_VEL
LIN {X 0,Y 523.457,Z 431.301,A -85,B 0,C 180,E1 24804.231,E2 24804.231} C_VEL
LIN {X 0,Y 527.948,Z 441.033,A -85,B 0,C 180,E1 24802.285,E2 24802.285} C_VEL
LIN {X 0,Y 529.954,Z 445.038,A -85,B 0,C 180,E1 24801.561,E2 24801.561} C_VEL
LIN {X 0,Y 540.872,Z 460.812,A -85,B 0,C 180,E1 24799.734,E2 24799.734} C_VEL
LIN {X 0,Y 551.915,Z 477.325,A -85,B 0,C 180,E1 24798.03,E2 24798.03} C_VEL
LIN {X 0,Y 565.109,Z 498.779,A -85,B 0,C 180,E1 24796.12,E2 24796.12} C_VEL
LIN {X 0,Y 571.456,Z 510.293,A -85,B 0,C 180,E1 24795.234,E2 24795.234} C_VEL
LIN {X 0,Y 564.184,Z 739.202,A -85,B 0,C 180,E1 24791.974,E2 24791.974} C_VEL
LIN {X 0,Y 561.026,Z 839.149,A -85,B 0,C 180,E1 24790.539,E2 24790.539} C_VEL
LIN {X 0,Y 559.226,Z 865.119,A -85,B 0,C 180,E1 24790.008,E2 24790.008} C_VEL
LIN {X 0,Y 557.22,Z 886.749,A -85,B 0,C 180,E1 24789.412,E2 24789.412} C_VEL
LIN {X 0,Y 554.443,Z 911.605,A -85,B 0,C 180,E1 24788.531,E2 24788.531} C_VEL
LIN {X 0,Y 551.817,Z 931.99,A -85,B 0,C 180,E1 24787.636,E2 24787.636} C_VEL
LIN {X 0,Y 548.583,Z 954.661,A -85,B 0,C 180,E1 24786.455,E2 24786.455} C_VEL
LIN {X 0,Y 545.454,Z 974.539,A -85,B 0,C 180,E1 24785.217,E2 24785.217} C_VEL
LIN {X 0,Y 542.266,Z 993.815,A -85,B 0,C 180,E1 24783.839,E2 24783.839} C_VEL
LIN {X 0,Y 538.663,Z 1014.374,A -85,B 0,C 180,E1 24782.128,E2 24782.128} C_VEL
LIN {X 0,Y 535.659,Z 1031.292,A -85,B 0,C 180,E1 24780.513,E2 24780.513} C_VEL
LIN {X 0,Y 532.244,Z 1050.719,A -85,B 0,C 180,E1 24778.379,E2 24778.379} C_VEL
LIN {X 0,Y 529.597,Z 1065.921,A -85,B 0,C 180,E1 24776.46,E2 24776.46} C_VEL
LIN {X 0,Y 526.91,Z 1082.383,A -85,B 0,C 180,E1 24774.079,E2 24774.079} C_VEL
LIN {X 0,Y 524.929,Z 1095.295,A -85,B 0,C 180,E1 24771.922,E2 24771.922} C_VEL
LIN {X 0,Y 523.163,Z 1108.327,A -85,B 0,C 180,E1 24769.424,E2 24769.424} C_VEL
LIN {X 0,Y 521.923,Z 1118.864,A -85,B 0,C 180,E1 24767.045,E2 24767.045} C_VEL
LIN {X 0,Y 520.989,Z 1128.726,A -85,B 0,C 180,E1 24764.448,E2 24764.448} C_VEL
LIN {X 0,Y 520.429,Z 1136.323,A -85,B 0,C 180,E1 24761.976,E2 24761.976} C_VEL
LIN {X 0,Y 520.136,Z 1142.249,A -85,B 0,C 180,E1 24759.628,E2 24759.628} C_VEL
LIN {X 0,Y 519.975,Z 1147.552,A -85,B 0,C 180,E1 24756.847,E2 24756.847} C_VEL
LIN {X 0,Y 519.937,Z 1150.576,A -85,B 0,C 180,E1 24754.522,E2 24754.522} C_VEL
LIN {X 0,Y 519.932,Z 1152.473,A -85,B 0,C 180,E1 24752.094,E2 24752.094} C_VEL
LIN {X 0,Y 519.912,Z 1152.911,A -85,B 0,C 180,E1 24749.449,E2 24749.449} C_VEL
LIN {X 0,Y 519.909,Z 1152.06,A -85,B 0,C 180,E1 24747.244,E2 24747.244} C_VEL
LIN {X 0,Y 519.918,Z 1150.003,A -85,B 0,C 180,E1 24744.925,E2 24744.925} C_VEL
LIN {X 0,Y 519.984,Z 1146.082,A -85,B 0,C 180,E1 24742.264,E2 24742.264} C_VEL
LIN {X 0,Y 520.17,Z 1141.236,A -85,B 0,C 180,E1 24739.926,E2 24739.926} C_VEL
LIN {X 0,Y 520.54,Z 1134.804,A -85,B 0,C 180,E1 24737.464,E2 24737.464} C_VEL
LIN {X 0,Y 521.203,Z 1126.292,A -85,B 0,C 180,E1 24734.876,E2 24734.876} C_VEL
LIN {X 0,Y 522.078,Z 1117.458,A -85,B 0,C 180,E1 24732.616,E2 24732.616} C_VEL
LIN {X 0,Y 523.587,Z 1104.862,A -85,B 0,C 180,E1 24729.895,E2 24729.895} C_VEL
LIN {X 0,Y 525.197,Z 1093.18,A -85,B 0,C 180,E1 24727.737,E2 24727.737} C_VEL
LIN {X 0,Y 527.452,Z 1078.342,A -85,B 0,C 180,E1 24725.351,E2 24725.351} C_VEL
LIN {X 0,Y 529.815,Z 1063.655,A -85,B 0,C 180,E1 24723.31,E2 24723.31} C_VEL
LIN {X 0,Y 532.69,Z 1046.701,A -85,B 0,C 180,E1 24721.234,E2 24721.234} C_VEL
LIN {X 0,Y 535.689,Z 1028.983,A -85,B 0,C 180,E1 24719.365,E2 24719.365} C_VEL
LIN {X 0,Y 539.012,Z 1009.735,A -85,B 0,C 180,E1 24717.581,E2 24717.581} C_VEL
LIN {X 0,Y 542.26,Z 989.725,A -85,B 0,C 180,E1 24715.996,E2 24715.996} C_VEL
LIN {X 0,Y 545.598,Z 968.702,A -85,B 0,C 180,E1 24714.547,E2 24714.547} C_VEL
LIN {X 0,Y 548.697,Z 947.055,A -85,B 0,C 180,E1 24713.293,E2 24713.293} C_VEL
LIN {X 0,Y 551.491,Z 926.339,A -85,B 0,C 180,E1 24712.272,E2 24712.272} C_VEL
LIN {X 0,Y 554.301,Z 902.185,A -85,B 0,C 180,E1 24711.293,E2 24711.293} C_VEL
LIN {X 0,Y 556.348,Z 881.837,A -85,B 0,C 180,E1 24710.627,E2 24710.627} C_VEL
LIN {X 0,Y 558.423,Z 857.011,A -85,B 0,C 180,E1 24709.994,E2 24709.994} C_VEL
LIN {X 0,Y 559.687,Z 833.948,A -85,B 0,C 180,E1 24709.571,E2 24709.571} C_VEL
LIN {X 0,Y 566.288,Z 602.803,A -85,B 0,C 180,E1 24706.317,E2 24706.317} C_VEL
LIN {X 0,Y 568.976,Z 508.989,A -85,B 0,C 180,E1 24704.983,E2 24704.983} C_VEL
LIN {X 0,Y 555.654,Z 485.882,A -85,B 0,C 180,E1 24703.248,E2 24703.248} C_VEL
LIN {X 0,Y 544.156,Z 467.292,A -85,B 0,C 180,E1 24701.661,E2 24701.661} C_VEL
LIN {X 0,Y 532.577,Z 449.793,A -85,B 0,C 180,E1 24699.966,E2 24699.966} C_VEL
LIN {X 0,Y 529.387,Z 444.828,A -85,B 0,C 180,E1 24699.42,E2 24699.42} C_VEL
LIN {X 0,Y 524.96,Z 434.873,A -85,B 0,C 180,E1 24697.692,E2 24697.692} C_VEL
LIN {X 0,Y 522.963,Z 430.569,A -85,B 0,C 180,E1 24696.896,E2 24696.896} C_VEL
LIN {X 0,Y 521.73,Z 427.326,A -85,B 0,C 180,E1 24696.238,E2 24696.238} C_VEL
LIN {X 0,Y 521.745,Z 427.212,A -85,B 0,C 180,E1 24692.844,E2 24692.844} C_VEL
LIN {X 0,Y 521.747,Z 427.211,A -85,B 0,C 180,E1 24689.381,E2 24689.381} C_VEL
LIN {X 0,Y 521.731,Z 427.236,A -85,B 0,C 180,E1 24685.91,E2 24685.91} C_VEL
LIN {X 0,Y 521.747,Z 427.229,A -85,B 0,C 180,E1 24682.419,E2 24682.419} C_VEL
LIN {X 0,Y 521.734,Z 427.21,A -85,B 0,C 180,E1 24678.898,E2 24678.898} C_VEL
LIN {X 0,Y 521.748,Z 427.222,A -85,B 0,C 180,E1 24675.428,E2 24675.428} C_VEL
LIN {X 0,Y 521.741,Z 427.236,A -85,B 0,C 180,E1 24671.945,E2 24671.945} C_VEL
LIN {X 0,Y 521.729,Z 427.204,A -85,B 0,C 180,E1 24668.486,E2 24668.486} C_VEL
LIN {X 0,Y 521.727,Z 427.231,A -85,B 0,C 180,E1 24664.947,E2 24664.947} C_VEL
LIN {X 0,Y 521.746,Z 427.226,A -85,B 0,C 180,E1 24661.428,E2 24661.428} C_VEL
LIN {X 0,Y 521.737,Z 427.207,A -85,B 0,C 180,E1 24658.023,E2 24658.023} C_VEL
LIN {X 0,Y 521.712,Z 427.243,A -85,B 0,C 180,E1 24654.611,E2 24654.611} C_VEL
LIN {X 0,Y 521.742,Z 427.205,A -85,B 0,C 180,E1 24651.292,E2 24651.292} C_VEL
LIN {X 0,Y 521.724,Z 427.23,A -85,B 0,C 180,E1 24647.942,E2 24647.942} C_VEL
LIN {X 0,Y 521.703,Z 427.236,A -85,B 0,C 180,E1 24644.549,E2 24644.549} C_VEL
LIN {X 0,Y 521.742,Z 427.206,A -85,B 0,C 180,E1 24641.214,E2 24641.214} C_VEL
LIN {X 0,Y 521.704,Z 427.242,A -85,B 0,C 180,E1 24637.935,E2 24637.935} C_VEL
LIN {X 0,Y 521.691,Z 427.235,A -85,B 0,C 180,E1 24634.453,E2 24634.453} C_VEL
LIN {X 0,Y 521.748,Z 427.21,A -85,B 0,C 180,E1 24631.122,E2 24631.122} C_VEL
LIN {X 0,Y 521.682,Z 427.227,A -85,B 0,C 180,E1 24627.905,E2 24627.905} C_VEL
LIN {X 0,Y 521.679,Z 427.237,A -85,B 0,C 180,E1 24624.358,E2 24624.358} C_VEL
LIN {X 0,Y 521.747,Z 427.238,A -85,B 0,C 180,E1 24621.054,E2 24621.054} C_VEL
LIN {X 0,Y 521.709,Z 427.394,A -85,B 0,C 180,E1 24618.509,E2 24618.509} C_VEL
LIN {X 0,Y 522.08,Z 428.9,A -85,B 0,C 180,E1 24618.258,E2 24618.258} C_VEL
LIN {X 0,Y 524.058,Z 431.94,A -85,B 0,C 180,E1 24617.929,E2 24617.929} C_VEL
LIN {X 0,Y 525.879,Z 433.69,A -85,B 0,C 180,E1 24617.657,E2 24617.657} C_VEL
LIN {X 0,Y 528.611,Z 437.643,A -85,B 0,C 180,E1 24617.229,E2 24617.229} C_VEL
LIN {X 0,Y 530.079,Z 439.527,A -85,B 0,C 180,E1 24617.007,E2 24617.007} C_VEL
LIN {X 0,Y 542.021,Z 455.841,A -85,B 0,C 180,E1 24615.262,E2 24615.262} C_VEL
LIN {X 0,Y 553.956,Z 472.819,A -85,B 0,C 180,E1 24613.63,E2 24613.63} C_VEL
LIN {X 0,Y 566.667,Z 492.542,A -85,B 0,C 180,E1 24611.983,E2 24611.983} C_VEL
LIN {X 0,Y 569.214,Z 497.09,A -85,B 0,C 180,E1 24611.656,E2 24611.656} C_VEL
LIN {X 0,Y 561.932,Z 743.819,A -85,B 0,C 180,E1 24608.189,E2 24608.189} C_VEL
LIN {X 0,Y 559.894,Z 810.012,A -85,B 0,C 180,E1 24607.239,E2 24607.239} C_VEL
LIN {X 0,Y 558.381,Z 834.747,A -85,B 0,C 180,E1 24606.714,E2 24606.714} C_VEL
LIN {X 0,Y 556.647,Z 855.872,A -85,B 0,C 180,E1 24606.119,E2 24606.119} C_VEL
LIN {X 0,Y 556.509,Z 857.594,A -85,B 0,C 180,E1 24606.065,E2 24606.065} C_VEL
LIN {X 0,Y 555.066,Z 865.043,A -85,B 0,C 180,E1 24605.882,E2 24605.882} C_VEL
LIN {X 0,Y 548.247,Z 883.715,A -85,B 0,C 180,E1 24605.552,E2 24605.552} C_VEL
LIN {X 0,Y 546.606,Z 890.898,A -85,B 0,C 180,E1 24605.314,E2 24605.314} C_VEL
LIN {X 0,Y 543.529,Z 913.618,A -85,B 0,C 180,E1 24604.195,E2 24604.195} C_VEL
LIN {X 0,Y 540.671,Z 933.058,A -85,B 0,C 180,E1 24603.063,E2 24603.063} C_VEL
LIN {X 0,Y 537.072,Z 955.221,A -85,B 0,C 180,E1 24601.544,E2 24601.544} C_VEL
LIN {X 0,Y 534.084,Z 972.41,A -85,B 0,C 180,E1 24600.177,E2 24600.177} C_VEL
LIN {X 0,Y 530.582,Z 991.792,A -85,B 0,C 180,E1 24598.414,E2 24598.414} C_VEL
LIN {X 0,Y 527.374,Z 1008.761,A -85,B 0,C 180,E1 24596.62,E2 24596.62} C_VEL
LIN {X 0,Y 524.239,Z 1025.79,A -85,B 0,C 180,E1 24594.57,E2 24594.57} C_VEL
LIN {X 0,Y 521.375,Z 1041.058,A -85,B 0,C 180,E1 24592.424,E2 24592.424} C_VEL
LIN {X 0,Y 518.934,Z 1055.116,A -85,B 0,C 180,E1 24590.176,E2 24590.176} C_VEL
LIN {X 0,Y 516.794,Z 1067.783,A -85,B 0,C 180,E1 24587.8,E2 24587.8} C_VEL
LIN {X 0,Y 515.242,Z 1078.285,A -85,B 0,C 180,E1 24585.534,E2 24585.534} C_VEL
LIN {X 0,Y 513.857,Z 1088.9,A -85,B 0,C 180,E1 24582.816,E2 24582.816} C_VEL
LIN {X 0,Y 513.073,Z 1096.283,A -85,B 0,C 180,E1 24580.556,E2 24580.556} C_VEL
LIN {X 0,Y 512.464,Z 1103.565,A -85,B 0,C 180,E1 24577.85,E2 24577.85} C_VEL
LIN {X 0,Y 512.145,Z 1108.772,A -85,B 0,C 180,E1 24575.31,E2 24575.31} C_VEL
LIN {X 0,Y 512.006,Z 1112.471,A -85,B 0,C 180,E1 24572.91,E2 24572.91} C_VEL
LIN {X 0,Y 511.971,Z 1115.161,A -85,B 0,C 180,E1 24570.112,E2 24570.112} C_VEL
LIN {X 0,Y 511.932,Z 1116.141,A -85,B 0,C 180,E1 24567.761,E2 24567.761} C_VEL
LIN {X 0,Y 511.919,Z 1115.957,A -85,B 0,C 180,E1 24565.182,E2 24565.182} C_VEL
LIN {X 0,Y 511.948,Z 1114.212,A -85,B 0,C 180,E1 24562.594,E2 24562.594} C_VEL
LIN {X 0,Y 512.016,Z 1111.57,A -85,B 0,C 180,E1 24560.332,E2 24560.332} C_VEL
LIN {X 0,Y 512.227,Z 1107.231,A -85,B 0,C 180,E1 24557.715,E2 24557.715} C_VEL
LIN {X 0,Y 512.647,Z 1101.164,A -85,B 0,C 180,E1 24555.081,E2 24555.081} C_VEL
LIN {X 0,Y 513.305,Z 1094.26,A -85,B 0,C 180,E1 24552.65,E2 24552.65} C_VEL
LIN {X 0,Y 514.468,Z 1084.439,A -85,B 0,C 180,E1 24549.84,E2 24549.84} C_VEL
LIN {X 0,Y 515.797,Z 1074.921,A -85,B 0,C 180,E1 24547.549,E2 24547.549} C_VEL
LIN {X 0,Y 517.912,Z 1061.82,A -85,B 0,C 180,E1 24544.866,E2 24544.866} C_VEL
LIN {X 0,Y 520.026,Z 1049.894,A -85,B 0,C 180,E1 24542.766,E2 24542.766} C_VEL
LIN {X 0,Y 522.877,Z 1034.745,A -85,B 0,C 180,E1 24540.438,E2 24540.438} C_VEL
LIN {X 0,Y 525.79,Z 1019.57,A -85,B 0,C 180,E1 24538.426,E2 24538.426} C_VEL
LIN {X 0,Y 529.275,Z 1002.06,A -85,B 0,C 180,E1 24536.391,E2 24536.391} C_VEL
LIN {X 0,Y 532.665,Z 984.259,A -85,B 0,C 180,E1 24534.613,E2 24534.613} C_VEL
LIN {X 0,Y 536.292,Z 965.127,A -85,B 0,C 180,E1 24532.939,E2 24532.939} C_VEL
LIN {X 0,Y 539.838,Z 944.94,A -85,B 0,C 180,E1 24531.438,E2 24531.438} C_VEL
LIN {X 0,Y 542.974,Z 925.97,A -85,B 0,C 180,E1 24530.214,E2 24530.214} C_VEL
LIN {X 0,Y 546.312,Z 903.649,A -85,B 0,C 180,E1 24528.993,E2 24528.993} C_VEL
LIN {X 0,Y 548.862,Z 884.433,A -85,B 0,C 180,E1 24528.112,E2 24528.112} C_VEL
LIN {X 0,Y 551.336,Z 863.134,A -85,B 0,C 180,E1 24527.291,E2 24527.291} C_VEL
LIN {X 0,Y 553.556,Z 839.196,A -85,B 0,C 180,E1 24526.568,E2 24526.568} C_VEL
LIN {X 0,Y 555.052,Z 818.679,A -85,B 0,C 180,E1 24526.092,E2 24526.092} C_VEL
LIN {X 0,Y 556.377,Z 789.17,A -85,B 0,C 180,E1 24525.603,E2 24525.603} C_VEL
LIN {X 0,Y 564.552,Z 541.549,A -85,B 0,C 180,E1 24522.061,E2 24522.061} C_VEL
LIN {X 0,Y 565.821,Z 500.887,A -85,B 0,C 180,E1 24521.459,E2 24521.459} C_VEL
LIN {X 0,Y 556.427,Z 486.424,A -85,B 0,C 180,E1 24520.141,E2 24520.141} C_VEL
LIN {X 0,Y 544.779,Z 469.693,A -85,B 0,C 180,E1 24518.41,E2 24518.41} C_VEL
LIN {X 0,Y 534.186,Z 455.454,A -85,B 0,C 180,E1 24516.73,E2 24516.73} C_VEL
LIN {X 0,Y 529.427,Z 449.298,A -85,B 0,C 180,E1 24515.937,E2 24515.937} C_VEL
LIN {X 0,Y 526.358,Z 445.234,A -85,B 0,C 180,E1 24515.408,E2 24515.408} C_VEL
LIN {X 0,Y 523.054,Z 441.004,A -85,B 0,C 180,E1 24514.827,E2 24514.827} C_VEL
LIN {X 0,Y 521.87,Z 439.557,A -85,B 0,C 180,E1 24514.617,E2 24514.617} C_VEL
LIN {X 0,Y 518.936,Z 436.003,A -85,B 0,C 180,E1 24514.088,E2 24514.088} C_VEL
LIN {X 0,Y 518.014,Z 434.359,A -85,B 0,C 180,E1 24513.907,E2 24513.907} C_VEL
LIN {X 0,Y 515.235,Z 431.961,A -85,B 0,C 180,E1 24513.412,E2 24513.412} C_VEL
LIN {X 0,Y 513.944,Z 429.132,A -85,B 0,C 180,E1 24513.103,E2 24513.103} C_VEL
LIN {X 0,Y 513.796,Z 428.243,A -85,B 0,C 180,E1 24512.753,E2 24512.753} C_VEL
LIN {X 0,Y 513.738,Z 428.134,A -85,B 0,C 180,E1 24509.5,E2 24509.5} C_VEL
LIN {X 0,Y 513.751,Z 428.237,A -85,B 0,C 180,E1 24505.95,E2 24505.95} C_VEL
LIN {X 0,Y 513.806,Z 428.225,A -85,B 0,C 180,E1 24502.543,E2 24502.543} C_VEL
LIN {X 0,Y 513.78,Z 428.214,A -85,B 0,C 180,E1 24499.084,E2 24499.084} C_VEL
LIN {X 0,Y 513.757,Z 428.204,A -85,B 0,C 180,E1 24495.696,E2 24495.696} C_VEL
LIN {X 0,Y 513.803,Z 428.208,A -85,B 0,C 180,E1 24492.332,E2 24492.332} C_VEL
LIN {X 0,Y 513.799,Z 428.23,A -85,B 0,C 180,E1 24488.844,E2 24488.844} C_VEL
LIN {X 0,Y 513.771,Z 428.218,A -85,B 0,C 180,E1 24485.472,E2 24485.472} C_VEL
LIN {X 0,Y 513.796,Z 428.195,A -85,B 0,C 180,E1 24482.007,E2 24482.007} C_VEL
LIN {X 0,Y 513.806,Z 428.21,A -85,B 0,C 180,E1 24478.55,E2 24478.55} C_VEL
LIN {X 0,Y 513.787,Z 428.225,A -85,B 0,C 180,E1 24475.088,E2 24475.088} C_VEL
LIN {X 0,Y 513.795,Z 428.204,A -85,B 0,C 180,E1 24471.607,E2 24471.607} C_VEL
LIN {X 0,Y 513.798,Z 428.199,A -85,B 0,C 180,E1 24468.204,E2 24468.204} C_VEL
LIN {X 0,Y 513.807,Z 428.218,A -85,B 0,C 180,E1 24464.653,E2 24464.653} C_VEL
LIN {X 0,Y 513.799,Z 428.231,A -85,B 0,C 180,E1 24461.049,E2 24461.049} C_VEL
LIN {X 0,Y 513.811,Z 428.189,A -85,B 0,C 180,E1 24457.457,E2 24457.457} C_VEL
LIN {X 0,Y 513.788,Z 428.195,A -85,B 0,C 180,E1 24454.031,E2 24454.031} C_VEL
LIN {X 0,Y 513.81,Z 428.225,A -85,B 0,C 180,E1 24450.505,E2 24450.505} C_VEL
LIN {X 0,Y 513.808,Z 428.217,A -85,B 0,C 180,E1 24446.983,E2 24446.983} C_VEL
LIN {X 0,Y 513.848,Z 428.62,A -85,B 0,C 180,E1 24446.151,E2 24446.151} C_VEL
LIN {X 0,Y 515.426,Z 432.153,A -85,B 0,C 180,E1 24445.361,E2 24445.361} C_VEL
LIN {X 0,Y 520.346,Z 442.612,A -85,B 0,C 180,E1 24443.163,E2 24443.163} C_VEL
LIN {X 0,Y 521.812,Z 445.172,A -85,B 0,C 180,E1 24442.734,E2 24442.734} C_VEL
LIN {X 0,Y 532.356,Z 459.924,A -85,B 0,C 180,E1 24440.887,E2 24440.887} C_VEL
LIN {X 0,Y 544.74,Z 478.439,A -85,B 0,C 180,E1 24438.884,E2 24438.884} C_VEL
LIN {X 0,Y 555.904,Z 496.217,A -85,B 0,C 180,E1 24437.199,E2 24437.199} C_VEL
LIN {X 0,Y 565.816,Z 513.584,A -85,B 0,C 180,E1 24435.773,E2 24435.773} C_VEL
LIN {X 0,Y 558.258,Z 741.606,A -85,B 0,C 180,E1 24432.499,E2 24432.499} C_VEL
LIN {X 0,Y 555.046,Z 838.876,A -85,B 0,C 180,E1 24431.091,E2 24431.091} C_VEL
LIN {X 0,Y 553.188,Z 864.837,A -85,B 0,C 180,E1 24430.557,E2 24430.557} C_VEL
LIN {X 0,Y 551.131,Z 886.247,A -85,B 0,C 180,E1 24429.964,E2 24429.964} C_VEL
LIN {X 0,Y 548.241,Z 911.118,A -85,B 0,C 180,E1 24429.081,E2 24429.081} C_VEL
LIN {X 0,Y 545.435,Z 932.048,A -85,B 0,C 180,E1 24428.155,E2 24428.155} C_VEL
LIN {X 0,Y 542.061,Z 954.643,A -85,B 0,C 180,E1 24426.966,E2 24426.966} C_VEL
LIN {X 0,Y 538.643,Z 975.436,A -85,B 0,C 180,E1 24425.654,E2 24425.654} C_VEL
LIN {X 0,Y 535.107,Z 995.941,A -85,B 0,C 180,E1 24424.16,E2 24424.16} C_VEL
LIN {X 0,Y 531.481,Z 1015.476,A -85,B 0,C 180,E1 24422.488,E2 24422.488} C_VEL
LIN {X 0,Y 528.163,Z 1033.388,A -85,B 0,C 180,E1 24420.74,E2 24420.74} C_VEL
LIN {X 0,Y 524.794,Z 1051.481,A -85,B 0,C 180,E1 24418.694,E2 24418.694} C_VEL
LIN {X 0,Y 522.039,Z 1066.586,A -85,B 0,C 180,E1 24416.751,E2 24416.751} C_VEL
LIN {X 0,Y 519.224,Z 1082.879,A -85,B 0,C 180,E1 24414.337,E2 24414.337} C_VEL
LIN {X 0,Y 517.156,Z 1095.712,A -85,B 0,C 180,E1 24412.149,E2 24412.149} C_VEL
LIN {X 0,Y 515.229,Z 1109.128,A -85,B 0,C 180,E1 24409.499,E2 24409.499} C_VEL
LIN {X 0,Y 514.006,Z 1119.075,A -85,B 0,C 180,E1 24407.199,E2 24407.199} C_VEL
LIN {X 0,Y 513.029,Z 1128.817,A -85,B 0,C 180,E1 24404.562,E2 24404.562} C_VEL
LIN {X 0,Y 512.444,Z 1136.354,A -85,B 0,C 180,E1 24402.051,E2 24402.051} C_VEL
LIN {X 0,Y 512.127,Z 1142.484,A -85,B 0,C 180,E1 24399.553,E2 24399.553} C_VEL
LIN {X 0,Y 511.976,Z 1147.428,A -85,B 0,C 180,E1 24396.842,E2 24396.842} C_VEL
LIN {X 0,Y 511.94,Z 1150.406,A -85,B 0,C 180,E1 24394.481,E2 24394.481} C_VEL
LIN {X 0,Y 511.932,Z 1152.325,A -85,B 0,C 180,E1 24391.903,E2 24391.903} C_VEL
LIN {X 0,Y 511.917,Z 1152.604,A -85,B 0,C 180,E1 24389.329,E2 24389.329} C_VEL
LIN {X 0,Y 511.912,Z 1151.706,A -85,B 0,C 180,E1 24387.089,E2 24387.089} C_VEL
LIN {X 0,Y 511.922,Z 1149.484,A -85,B 0,C 180,E1 24384.62,E2 24384.62} C_VEL
LIN {X 0,Y 512.013,Z 1145.372,A -85,B 0,C 180,E1 24381.917,E2 24381.917} C_VEL
LIN {X 0,Y 512.198,Z 1140.682,A -85,B 0,C 180,E1 24379.654,E2 24379.654} C_VEL
LIN {X 0,Y 512.631,Z 1133.86,A -85,B 0,C 180,E1 24377.038,E2 24377.038} C_VEL
LIN {X 0,Y 513.327,Z 1125.559,A -85,B 0,C 180,E1 24374.523,E2 24374.523} C_VEL
LIN {X 0,Y 514.332,Z 1116.189,A -85,B 0,C 180,E1 24372.112,E2 24372.112} C_VEL
LIN {X 0,Y 515.811,Z 1104.511,A -85,B 0,C 180,E1 24369.578,E2 24369.578} C_VEL
LIN {X 0,Y 517.526,Z 1092.816,A -85,B 0,C 180,E1 24367.388,E2 24367.388} C_VEL
LIN {X 0,Y 519.945,Z 1077.671,A -85,B 0,C 180,E1 24364.927,E2 24364.927} C_VEL
LIN {X 0,Y 522.435,Z 1063.025,A -85,B 0,C 180,E1 24362.87,E2 24362.87} C_VEL
LIN {X 0,Y 525.512,Z 1045.626,A -85,B 0,C 180,E1 24360.725,E2 24360.725} C_VEL
LIN {X 0,Y 528.564,Z 1028.534,A -85,B 0,C 180,E1 24358.906,E2 24358.906} C_VEL
LIN {X 0,Y 532.031,Z 1009.251,A -85,B 0,C 180,E1 24357.102,E2 24357.102} C_VEL
LIN {X 0,Y 535.35,Z 989.646,A -85,B 0,C 180,E1 24355.533,E2 24355.533} C_VEL
LIN {X 0,Y 538.769,Z 968.991,A -85,B 0,C 180,E1 24354.094,E2 24354.094} C_VEL
LIN {X 0,Y 541.996,Z 947.479,A -85,B 0,C 180,E1 24352.83,E2 24352.83} C_VEL
LIN {X 0,Y 544.726,Z 927.992,A -85,B 0,C 180,E1 24351.853,E2 24351.853} C_VEL
LIN {X 0,Y 547.75,Z 903.423,A -85,B 0,C 180,E1 24350.831,E2 24350.831} C_VEL
LIN {X 0,Y 549.918,Z 882.761,A -85,B 0,C 180,E1 24350.142,E2 24350.142} C_VEL
LIN {X 0,Y 552.064,Z 858.702,A -85,B 0,C 180,E1 24349.51,E2 24349.51} C_VEL
LIN {X 0,Y 553.464,Z 834.376,A -85,B 0,C 180,E1 24349.055,E2 24349.055} C_VEL
LIN {X 0,Y 560.347,Z 603.705,A -85,B 0,C 180,E1 24345.779,E2 24345.779} C_VEL
LIN {X 0,Y 563.104,Z 512.19,A -85,B 0,C 180,E1 24344.468,E2 24344.468} C_VEL
LIN {X 0,Y 550.368,Z 490.134,A -85,B 0,C 180,E1 24342.767,E2 24342.767} C_VEL
LIN {X 0,Y 537.748,Z 469.57,A -85,B 0,C 180,E1 24340.971,E2 24340.971} C_VEL
LIN {X 0,Y 525.68,Z 451.504,A -85,B 0,C 180,E1 24339.143,E2 24339.143} C_VEL
LIN {X 0,Y 521.11,Z 444.558,A -85,B 0,C 180,E1 24338.369,E2 24338.369} C_VEL
LIN {X 0,Y 516.561,Z 434.972,A -85,B 0,C 180,E1 24336.597,E2 24336.597} C_VEL
LIN {X 0,Y 514.895,Z 431.397,A -85,B 0,C 180,E1 24335.907,E2 24335.907} C_VEL
LIN {X 0,Y 513.829,Z 428.377,A -85,B 0,C 180,E1 24335.307,E2 24335.307} C_VEL
LIN {X 0,Y 513.79,Z 428.213,A -85,B 0,C 180,E1 24331.83,E2 24331.83} C_VEL
LIN {X 0,Y 513.796,Z 428.197,A -85,B 0,C 180,E1 24328.349,E2 24328.349} C_VEL
LIN {X 0,Y 513.801,Z 428.198,A -85,B 0,C 180,E1 24324.857,E2 24324.857} C_VEL
LIN {X 0,Y 513.809,Z 428.229,A -85,B 0,C 180,E1 24321.341,E2 24321.341} C_VEL
LIN {X 0,Y 513.796,Z 428.214,A -85,B 0,C 180,E1 24317.79,E2 24317.79} C_VEL
LIN {X 0,Y 513.809,Z 428.192,A -85,B 0,C 180,E1 24314.273,E2 24314.273} C_VEL
LIN {X 0,Y 513.791,Z 428.226,A -85,B 0,C 180,E1 24310.768,E2 24310.768} C_VEL
LIN {X 0,Y 513.806,Z 428.207,A -85,B 0,C 180,E1 24307.267,E2 24307.267} C_VEL
LIN {X 0,Y 513.801,Z 428.195,A -85,B 0,C 180,E1 24303.794,E2 24303.794} C_VEL
LIN {X 0,Y 513.787,Z 428.23,A -85,B 0,C 180,E1 24300.335,E2 24300.335} C_VEL
LIN {X 0,Y 513.776,Z 428.199,A -85,B 0,C 180,E1 24296.765,E2 24296.765} C_VEL
LIN {X 0,Y 513.813,Z 428.207,A -85,B 0,C 180,E1 24293.295,E2 24293.295} C_VEL
LIN {X 0,Y 513.799,Z 428.223,A -85,B 0,C 180,E1 24289.799,E2 24289.799} C_VEL
LIN {X 0,Y 513.76,Z 428.195,A -85,B 0,C 180,E1 24286.379,E2 24286.379} C_VEL
LIN {X 0,Y 513.784,Z 428.224,A -85,B 0,C 180,E1 24282.91,E2 24282.91} C_VEL
LIN {X 0,Y 513.804,Z 428.216,A -85,B 0,C 180,E1 24279.495,E2 24279.495} C_VEL
LIN {X 0,Y 513.749,Z 428.198,A -85,B 0,C 180,E1 24276.17,E2 24276.17} C_VEL
LIN {X 0,Y 513.775,Z 428.22,A -85,B 0,C 180,E1 24272.784,E2 24272.784} C_VEL
LIN {X 0,Y 513.781,Z 428.23,A -85,B 0,C 180,E1 24269.473,E2 24269.473} C_VEL
LIN {X 0,Y 513.737,Z 428.217,A -85,B 0,C 180,E1 24266.176,E2 24266.176} C_VEL
LIN {X 0,Y 513.782,Z 428.206,A -85,B 0,C 180,E1 24262.893,E2 24262.893} C_VEL
LIN {X 0,Y 513.742,Z 428.26,A -85,B 0,C 180,E1 24259.673,E2 24259.673} C_VEL
LIN {X 0,Y 513.937,Z 429.147,A -85,B 0,C 180,E1 24259.39,E2 24259.39} C_VEL
LIN {X 0,Y 515.773,Z 432.492,A -85,B 0,C 180,E1 24259.024,E2 24259.024} C_VEL
LIN {X 0,Y 517.945,Z 434.619,A -85,B 0,C 180,E1 24258.682,E2 24258.682} C_VEL
LIN {X 0,Y 520.459,Z 438.428,A -85,B 0,C 180,E1 24258.265,E2 24258.265} C_VEL
LIN {X 0,Y 522.42,Z 440.669,A -85,B 0,C 180,E1 24257.96,E2 24257.96} C_VEL
LIN {X 0,Y 534.176,Z 456.643,A -85,B 0,C 180,E1 24256.165,E2 24256.165} C_VEL
LIN {X 0,Y 544.649,Z 471.38,A -85,B 0,C 180,E1 24254.67,E2 24254.67} C_VEL
LIN {X 0,Y 557.855,Z 491.176,A -85,B 0,C 180,E1 24252.892,E2 24252.892} C_VEL
LIN {X 0,Y 563.341,Z 500.486,A -85,B 0,C 180,E1 24252.173,E2 24252.173} C_VEL
LIN {X 0,Y 555.773,Z 746.25,A -85,B 0,C 180,E1 24248.69,E2 24248.69} C_VEL
LIN {X 0,Y 553.707,Z 810.457,A -85,B 0,C 180,E1 24247.759,E2 24247.759} C_VEL
LIN {X 0,Y 552.14,Z 835.113,A -85,B 0,C 180,E1 24247.231,E2 24247.231} C_VEL
LIN {X 0,Y 550.328,Z 856.441,A -85,B 0,C 180,E1 24246.625,E2 24246.625} C_VEL
LIN {X 0,Y 547.798,Z 880.807,A -85,B 0,C 180,E1 24245.739,E2 24245.739} C_VEL
LIN {X 0,Y 546.606,Z 890.898,A -85,B 0,C 180,E1 24245.314,E2 24245.314} C_VEL
LIN {X 0,Y 544.934,Z 898.088,A -85,B 0,C 180,E1 24245.059,E2 24245.059} C_VEL
LIN {X 0,Y 537.586,Z 916.12,A -85,B 0,C 180,E1 24244.525,E2 24244.525} C_VEL
LIN {X 0,Y 535.739,Z 922.985,A -85,B 0,C 180,E1 24244.197,E2 24244.197} C_VEL
LIN {X 0,Y 532.362,Z 943.69,A -85,B 0,C 180,E1 24242.875,E2 24242.875} C_VEL
LIN {X 0,Y 528.991,Z 963.106,A -85,B 0,C 180,E1 24241.446,E2 24241.446} C_VEL
LIN {X 0,Y 525.259,Z 983.031,A -85,B 0,C 180,E1 24239.729,E2 24239.729} C_VEL
LIN {X 0,Y 522.018,Z 999.991,A -85,B 0,C 180,E1 24238.05,E2 24238.05} C_VEL
LIN {X 0,Y 518.439,Z 1018.233,A -85,B 0,C 180,E1 24235.964,E2 24235.964} C_VEL
LIN {X 0,Y 515.508,Z 1033.193,A -85,B 0,C 180,E1 24233.997,E2 24233.997} C_VEL
LIN {X 0,Y 512.424,Z 1049.468,A -85,B 0,C 180,E1 24231.521,E2 24231.521} C_VEL
LIN {X 0,Y 510.186,Z 1061.829,A -85,B 0,C 180,E1 24229.343,E2 24229.343} C_VEL
LIN {X 0,Y 507.974,Z 1075.228,A -85,B 0,C 180,E1 24226.584,E2 24226.584} C_VEL
LIN {X 0,Y 506.604,Z 1084.714,A -85,B 0,C 180,E1 24224.281,E2 24224.281} C_VEL
LIN {X 0,Y 505.425,Z 1094.284,A -85,B 0,C 180,E1 24221.526,E2 24221.526} C_VEL
LIN {X 0,Y 504.711,Z 1101.389,A -85,B 0,C 180,E1 24219.004,E2 24219.004} C_VEL
LIN {X 0,Y 504.253,Z 1107.605,A -85,B 0,C 180,E1 24216.261,E2 24216.261} C_VEL
LIN {X 0,Y 504.029,Z 1111.881,A -85,B 0,C 180,E1 24213.64,E2 24213.64} C_VEL
LIN {X 0,Y 503.959,Z 1114.496,A -85,B 0,C 180,E1 24211.364,E2 24211.364} C_VEL
LIN {X 0,Y 503.922,Z 1116.257,A -85,B 0,C 180,E1 24208.636,E2 24208.636} C_VEL
LIN {X 0,Y 503.933,Z 1116.429,A -85,B 0,C 180,E1 24206.132,E2 24206.132} C_VEL
LIN {X 0,Y 503.964,Z 1115.45,A -85,B 0,C 180,E1 24203.728,E2 24203.728} C_VEL
LIN {X 0,Y 504.018,Z 1112.739,A -85,B 0,C 180,E1 24200.868,E2 24200.868} C_VEL
LIN {X 0,Y 504.176,Z 1109.061,A -85,B 0,C 180,E1 24198.44,E2 24198.44} C_VEL
LIN {X 0,Y 504.548,Z 1103.694,A -85,B 0,C 180,E1 24195.774,E2 24195.774} C_VEL
LIN {X 0,Y 505.203,Z 1096.559,A -85,B 0,C 180,E1 24193.086,E2 24193.086} C_VEL
LIN {X 0,Y 506.092,Z 1089.029,A -85,B 0,C 180,E1 24190.735,E2 24190.735} C_VEL
LIN {X 0,Y 507.657,Z 1078.117,A -85,B 0,C 180,E1 24187.902,E2 24187.902} C_VEL
LIN {X 0,Y 509.339,Z 1067.781,A -85,B 0,C 180,E1 24185.629,E2 24185.629} C_VEL
LIN {X 0,Y 511.832,Z 1054.165,A -85,B 0,C 180,E1 24183.049,E2 24183.049} C_VEL
LIN {X 0,Y 514.356,Z 1041.097,A -85,B 0,C 180,E1 24180.922,E2 24180.922} C_VEL
LIN {X 0,Y 517.552,Z 1025.457,A -85,B 0,C 180,E1 24178.688,E2 24178.688} C_VEL
LIN {X 0,Y 520.835,Z 1009.23,A -85,B 0,C 180,E1 24176.697,E2 24176.697} C_VEL
LIN {X 0,Y 524.47,Z 991.712,A -85,B 0,C 180,E1 24174.81,E2 24174.81} C_VEL
LIN {X 0,Y 528.207,Z 972.673,A -85,B 0,C 180,E1 24173.05,E2 24173.05} C_VEL
LIN {X 0,Y 531.697,Z 954.337,A -85,B 0,C 180,E1 24171.572,E2 24171.572} C_VEL
LIN {X 0,Y 535.605,Z 932.109,A -85,B 0,C 180,E1 24170.044,E2 24170.044} C_VEL
LIN {X 0,Y 538.77,Z 912.436,A -85,B 0,C 180,E1 24168.894,E2 24168.894} C_VEL
LIN {X 0,Y 542.141,Z 889.21,A -85,B 0,C 180,E1 24167.758,E2 24167.758} C_VEL
LIN {X 0,Y 544.584,Z 869.221,A -85,B 0,C 180,E1 24166.95,E2 24166.95} C_VEL
LIN {X 0,Y 547.082,Z 845.703,A -85,B 0,C 180,E1 24166.176,E2 24166.176} C_VEL
LIN {X 0,Y 548.894,Z 822.491,A -85,B 0,C 180,E1 24165.607,E2 24165.607} C_VEL
LIN {X 0,Y 550.114,Z 800.154,A -85,B 0,C 180,E1 24165.2,E2 24165.2} C_VEL
LIN {X 0,Y 558.75,Z 549.505,A -85,B 0,C 180,E1 24161.581,E2 24161.581} C_VEL
LIN {X 0,Y 560.274,Z 504.529,A -85,B 0,C 180,E1 24160.917,E2 24160.917} C_VEL
LIN {X 0,Y 548.071,Z 485.949,A -85,B 0,C 180,E1 24159.142,E2 24159.142} C_VEL
LIN {X 0,Y 537.21,Z 470.753,A -85,B 0,C 180,E1 24157.457,E2 24157.457} C_VEL
LIN {X 0,Y 529.671,Z 460.669,A -85,B 0,C 180,E1 24156.219,E2 24156.219} C_VEL
LIN {X 0,Y 522.867,Z 451.706,A -85,B 0,C 180,E1 24155.042,E2 24155.042} C_VEL
LIN {X 0,Y 518.421,Z 446.082,A -85,B 0,C 180,E1 24154.243,E2 24154.243} C_VEL
LIN {X 0,Y 515.226,Z 441.866,A -85,B 0,C 180,E1 24153.647,E2 24153.647} C_VEL
LIN {X 0,Y 511.51,Z 437.779,A -85,B 0,C 180,E1 24152.951,E2 24152.951} C_VEL
LIN {X 0,Y 510.209,Z 435.385,A -85,B 0,C 180,E1 24152.678,E2 24152.678} C_VEL
LIN {X 0,Y 507.266,Z 432.892,A -85,B 0,C 180,E1 24152.122,E2 24152.122} C_VEL
LIN {X 0,Y 505.963,Z 430.086,A -85,B 0,C 180,E1 24151.787,E2 24151.787} C_VEL
LIN {X 0,Y 505.814,Z 429.243,A -85,B 0,C 180,E1 24151.458,E2 24151.458} C_VEL
LIN {X 0,Y 505.798,Z 429.149,A -85,B 0,C 180,E1 24147.938,E2 24147.938} C_VEL
LIN {X 0,Y 505.861,Z 429.194,A -85,B 0,C 180,E1 24144.599,E2 24144.599} C_VEL
LIN {X 0,Y 505.822,Z 429.209,A -85,B 0,C 180,E1 24141.329,E2 24141.329} C_VEL
LIN {X 0,Y 505.825,Z 429.224,A -85,B 0,C 180,E1 24137.842,E2 24137.842} C_VEL
LIN {X 0,Y 505.874,Z 429.205,A -85,B 0,C 180,E1 24134.415,E2 24134.415} C_VEL
LIN {X 0,Y 505.848,Z 429.191,A -85,B 0,C 180,E1 24130.939,E2 24130.939} C_VEL
LIN {X 0,Y 505.828,Z 429.197,A -85,B 0,C 180,E1 24127.497,E2 24127.497} C_VEL
LIN {X 0,Y 505.861,Z 429.216,A -85,B 0,C 180,E1 24124.081,E2 24124.081} C_VEL
LIN {X 0,Y 505.869,Z 429.198,A -85,B 0,C 180,E1 24120.566,E2 24120.566} C_VEL
LIN {X 0,Y 505.843,Z 429.184,A -85,B 0,C 180,E1 24117.054,E2 24117.054} C_VEL
LIN {X 0,Y 505.851,Z 429.196,A -85,B 0,C 180,E1 24113.531,E2 24113.531} C_VEL
LIN {X 0,Y 505.867,Z 429.216,A -85,B 0,C 180,E1 24109.983,E2 24109.983} C_VEL
LIN {X 0,Y 505.864,Z 429.202,A -85,B 0,C 180,E1 24106.396,E2 24106.396} C_VEL
LIN {X 0,Y 505.856,Z 429.19,A -85,B 0,C 180,E1 24102.871,E2 24102.871} C_VEL
LIN {X 0,Y 505.863,Z 429.183,A -85,B 0,C 180,E1 24099.4,E2 24099.4} C_VEL
LIN {X 0,Y 505.856,Z 429.219,A -85,B 0,C 180,E1 24095.953,E2 24095.953} C_VEL
LIN {X 0,Y 505.863,Z 429.18,A -85,B 0,C 180,E1 24092.45,E2 24092.45} C_VEL
LIN {X 0,Y 505.864,Z 429.18,A -85,B 0,C 180,E1 24088.943,E2 24088.943} C_VEL
LIN {X 0,Y 505.9,Z 429.48,A -85,B 0,C 180,E1 24087.391,E2 24087.391} C_VEL
LIN {X 0,Y 507.504,Z 433.17,A -85,B 0,C 180,E1 24086.519,E2 24086.519} C_VEL
LIN {X 0,Y 510.5,Z 439.395,A -85,B 0,C 180,E1 24085.115,E2 24085.115} C_VEL
LIN {X 0,Y 512.705,Z 443.903,A -85,B 0,C 180,E1 24084.192,E2 24084.192} C_VEL
LIN {X 0,Y 523.435,Z 458.704,A -85,B 0,C 180,E1 24082.179,E2 24082.179} C_VEL
LIN {X 0,Y 535.601,Z 476.359,A -85,B 0,C 180,E1 24080.101,E2 24080.101} C_VEL
LIN {X 0,Y 548.078,Z 495.986,A -85,B 0,C 180,E1 24078.126,E2 24078.126} C_VEL
LIN {X 0,Y 558.522,Z 513.78,A -85,B 0,C 180,E1 24076.571,E2 24076.571} C_VEL
LIN {X 0,Y 560.215,Z 517.171,A -85,B 0,C 180,E1 24076.319,E2 24076.319} C_VEL
LIN {X 0,Y 552.404,Z 743.281,A -85,B 0,C 180,E1 24073.047,E2 24073.047} C_VEL
LIN {X 0,Y 549.119,Z 838.623,A -85,B 0,C 180,E1 24071.654,E2 24071.654} C_VEL
LIN {X 0,Y 547.201,Z 864.568,A -85,B 0,C 180,E1 24071.117,E2 24071.117} C_VEL
LIN {X 0,Y 545.106,Z 885.647,A -85,B 0,C 180,E1 24070.531,E2 24070.531} C_VEL
LIN {X 0,Y 542.325,Z 909.068,A -85,B 0,C 180,E1 24069.706,E2 24069.706} C_VEL
LIN {X 0,Y 539.337,Z 930.537,A -85,B 0,C 180,E1 24068.761,E2 24068.761} C_VEL
LIN {X 0,Y 535.903,Z 952.817,A -85,B 0,C 180,E1 24067.598,E2 24067.598} C_VEL
LIN {X 0,Y 532.167,Z 974.582,A -85,B 0,C 180,E1 24066.222,E2 24066.222} C_VEL
LIN {X 0,Y 528.47,Z 995.142,A -85,B 0,C 180,E1 24064.716,E2 24064.716} C_VEL
LIN {X 0,Y 524.65,Z 1014.925,A -85,B 0,C 180,E1 24063.011,E2 24063.011} C_VEL
LIN {X 0,Y 521.216,Z 1032.55,A -85,B 0,C 180,E1 24061.277,E2 24061.277} C_VEL
LIN {X 0,Y 517.592,Z 1051.038,A -85,B 0,C 180,E1 24059.169,E2 24059.169} C_VEL
LIN {X 0,Y 514.617,Z 1066.592,A -85,B 0,C 180,E1 24057.141,E2 24057.141} C_VEL
LIN {X 0,Y 511.675,Z 1082.674,A -85,B 0,C 180,E1 24054.72,E2 24054.72} C_VEL
LIN {X 0,Y 509.494,Z 1095.494,A -85,B 0,C 180,E1 24052.501,E2 24052.501} C_VEL
LIN {X 0,Y 507.452,Z 1108.891,A -85,B 0,C 180,E1 24049.811,E2 24049.811} C_VEL
LIN {X 0,Y 506.148,Z 1118.828,A -85,B 0,C 180,E1 24047.474,E2 24047.474} C_VEL
LIN {X 0,Y 505.108,Z 1128.556,A -85,B 0,C 180,E1 24044.795,E2 24044.795} C_VEL
LIN {X 0,Y 504.484,Z 1136.086,A -85,B 0,C 180,E1 24042.244,E2 24042.244} C_VEL
LIN {X 0,Y 504.141,Z 1142.246,A -85,B 0,C 180,E1 24039.69,E2 24039.69} C_VEL
LIN {X 0,Y 503.984,Z 1147.148,A -85,B 0,C 180,E1 24036.951,E2 24036.951} C_VEL
LIN {X 0,Y 503.941,Z 1150.123,A -85,B 0,C 180,E1 24034.552,E2 24034.552} C_VEL
LIN {X 0,Y 503.938,Z 1152.042,A -85,B 0,C 180,E1 24031.933,E2 24031.933} C_VEL
LIN {X 0,Y 503.922,Z 1152.318,A -85,B 0,C 180,E1 24029.318,E2 24029.318} C_VEL
LIN {X 0,Y 503.917,Z 1151.42,A -85,B 0,C 180,E1 24027.043,E2 24027.043} C_VEL
LIN {X 0,Y 503.928,Z 1149.195,A -85,B 0,C 180,E1 24024.535,E2 24024.535} C_VEL
LIN {X 0,Y 504.029,Z 1145.076,A -85,B 0,C 180,E1 24021.788,E2 24021.788} C_VEL
LIN {X 0,Y 504.219,Z 1140.379,A -85,B 0,C 180,E1 24019.488,E2 24019.488} C_VEL
LIN {X 0,Y 504.681,Z 1133.543,A -85,B 0,C 180,E1 24016.83,E2 24016.83} C_VEL
LIN {X 0,Y 505.42,Z 1125.231,A -85,B 0,C 180,E1 24014.274,E2 24014.274} C_VEL
LIN {X 0,Y 506.488,Z 1115.849,A -85,B 0,C 180,E1 24011.825,E2 24011.825} C_VEL
LIN {X 0,Y 508.097,Z 1103.84,A -85,B 0,C 180,E1 24009.19,E2 24009.19} C_VEL
LIN {X 0,Y 509.863,Z 1092.444,A -85,B 0,C 180,E1 24007.029,E2 24007.029} C_VEL
LIN {X 0,Y 512.505,Z 1076.773,A -85,B 0,C 180,E1 24004.458,E2 24004.458} C_VEL
LIN {X 0,Y 515.158,Z 1061.981,A -85,B 0,C 180,E1 24002.362,E2 24002.362} C_VEL
LIN {X 0,Y 518.654,Z 1043.123,A -85,B 0,C 180,E1 24000.045,E2 24000.045} C_VEL
LIN {X 0,Y 521.688,Z 1026.943,A -85,B 0,C 180,E1 23998.32,E2 23998.32} C_VEL
LIN {X 0,Y 525.356,Z 1007.135,A -85,B 0,C 180,E1 23996.474,E2 23996.474} C_VEL
LIN {X 0,Y 528.657,Z 988.543,A -85,B 0,C 180,E1 23994.982,E2 23994.982} C_VEL
LIN {X 0,Y 532.285,Z 967.52,A -85,B 0,C 180,E1 23993.513,E2 23993.513} C_VEL
LIN {X 0,Y 535.488,Z 946.873,A -85,B 0,C 180,E1 23992.3,E2 23992.3} C_VEL
LIN {X 0,Y 538.488,Z 926.202,A -85,B 0,C 180,E1 23991.262,E2 23991.262} C_VEL
LIN {X 0,Y 541.541,Z 901.916,A -85,B 0,C 180,E1 23990.259,E2 23990.259} C_VEL
LIN {X 0,Y 543.707,Z 881.943,A -85,B 0,C 180,E1 23989.595,E2 23989.595} C_VEL
LIN {X 0,Y 545.904,Z 857.834,A -85,B 0,C 180,E1 23988.963,E2 23988.963} C_VEL
LIN {X 0,Y 547.322,Z 833.917,A -85,B 0,C 180,E1 23988.514,E2 23988.514} C_VEL
LIN {X 0,Y 554.481,Z 603.827,A -85,B 0,C 180,E1 23985.218,E2 23985.218} C_VEL
LIN {X 0,Y 557.192,Z 515.36,A -85,B 0,C 180,E1 23983.932,E2 23983.932} C_VEL
LIN {X 0,Y 543.785,Z 492,A -85,B 0,C 180,E1 23982.085,E2 23982.085} C_VEL
LIN {X 0,Y 529.516,Z 469.143,A -85,B 0,C 180,E1 23979.979,E2 23979.979} C_VEL
LIN {X 0,Y 516.261,Z 449.736,A -85,B 0,C 180,E1 23977.877,E2 23977.877} C_VEL
LIN {X 0,Y 512.517,Z 444.253,A -85,B 0,C 180,E1 23977.214,E2 23977.214} C_VEL
LIN {X 0,Y 508.826,Z 436.355,A -85,B 0,C 180,E1 23975.707,E2 23975.707} C_VEL
LIN {X 0,Y 507.245,Z 432.802,A -85,B 0,C 180,E1 23975.004,E2 23975.004} C_VEL
LIN {X 0,Y 505.864,Z 429.362,A -85,B 0,C 180,E1 23974.247,E2 23974.247} C_VEL
LIN {X 0,Y 505.876,Z 429.22,A -85,B 0,C 180,E1 23970.792,E2 23970.792} C_VEL
LIN {X 0,Y 505.868,Z 429.205,A -85,B 0,C 180,E1 23967.194,E2 23967.194} C_VEL
LIN {X 0,Y 505.856,Z 429.182,A -85,B 0,C 180,E1 23963.657,E2 23963.657} C_VEL
LIN {X 0,Y 505.858,Z 429.194,A -85,B 0,C 180,E1 23960.117,E2 23960.117} C_VEL
LIN {X 0,Y 505.866,Z 429.218,A -85,B 0,C 180,E1 23956.534,E2 23956.534} C_VEL
LIN {X 0,Y 505.853,Z 429.192,A -85,B 0,C 180,E1 23952.97,E2 23952.97} C_VEL
LIN {X 0,Y 505.861,Z 429.184,A -85,B 0,C 180,E1 23949.443,E2 23949.443} C_VEL
LIN {X 0,Y 505.869,Z 429.217,A -85,B 0,C 180,E1 23945.899,E2 23945.899} C_VEL
LIN {X 0,Y 505.845,Z 429.186,A -85,B 0,C 180,E1 23942.379,E2 23942.379} C_VEL
LIN {X 0,Y 505.844,Z 429.2,A -85,B 0,C 180,E1 23938.867,E2 23938.867} C_VEL
LIN {X 0,Y 505.868,Z 429.21,A -85,B 0,C 180,E1 23935.352,E2 23935.352} C_VEL
LIN {X 0,Y 505.862,Z 429.177,A -85,B 0,C 180,E1 23931.818,E2 23931.818} C_VEL
LIN {X 0,Y 505.83,Z 429.217,A -85,B 0,C 180,E1 23928.368,E2 23928.368} C_VEL
LIN {X 0,Y 505.84,Z 429.2,A -85,B 0,C 180,E1 23924.875,E2 23924.875} C_VEL
LIN {X 0,Y 505.865,Z 429.183,A -85,B 0,C 180,E1 23921.444,E2 23921.444} C_VEL
LIN {X 0,Y 505.82,Z 429.221,A -85,B 0,C 180,E1 23918.061,E2 23918.061} C_VEL
LIN {X 0,Y 505.814,Z 429.21,A -85,B 0,C 180,E1 23914.473,E2 23914.473} C_VEL
LIN {X 0,Y 505.86,Z 429.187,A -85,B 0,C 180,E1 23911.035,E2 23911.035} C_VEL
LIN {X 0,Y 505.812,Z 429.199,A -85,B 0,C 180,E1 23907.742,E2 23907.742} C_VEL
LIN {X 0,Y 505.8,Z 429.212,A -85,B 0,C 180,E1 23904.326,E2 23904.326} C_VEL
LIN {X 0,Y 505.852,Z 429.216,A -85,B 0,C 180,E1 23900.909,E2 23900.909} C_VEL
LIN {X 0,Y 505.886,Z 429.673,A -85,B 0,C 180,E1 23900.587,E2 23900.587} C_VEL
LIN {X 0,Y 506.582,Z 431.783,A -85,B 0,C 180,E1 23900.344,E2 23900.344} C_VEL
LIN {X 0,Y 508.884,Z 434.548,A -85,B 0,C 180,E1 23899.947,E2 23899.947} C_VEL
LIN {X 0,Y 510.231,Z 435.837,A -85,B 0,C 180,E1 23899.725,E2 23899.725} C_VEL
LIN {X 0,Y 512.907,Z 439.691,A -85,B 0,C 180,E1 23899.263,E2 23899.263} C_VEL
LIN {X 0,Y 514.535,Z 441.605,A -85,B 0,C 180,E1 23898.996,E2 23898.996} C_VEL
LIN {X 0,Y 517.858,Z 445.902,A -85,B 0,C 180,E1 23898.453,E2 23898.453} C_VEL
LIN {X 0,Y 530.371,Z 462.981,A -85,B 0,C 180,E1 23896.499,E2 23896.499} C_VEL
LIN {X 0,Y 542.365,Z 479.956,A -85,B 0,C 180,E1 23894.764,E2 23894.764} C_VEL
LIN {X 0,Y 556.826,Z 502.435,A -85,B 0,C 180,E1 23892.797,E2 23892.797} C_VEL
LIN {X 0,Y 557.512,Z 504.009,A -85,B 0,C 180,E1 23892.698,E2 23892.698} C_VEL
LIN {X 0,Y 549.657,Z 748.661,A -85,B 0,C 180,E1 23889.202,E2 23889.202} C_VEL
LIN {X 0,Y 547.564,Z 810.952,A -85,B 0,C 180,E1 23888.29,E2 23888.29} C_VEL
LIN {X 0,Y 545.935,Z 835.593,A -85,B 0,C 180,E1 23887.756,E2 23887.756} C_VEL
LIN {X 0,Y 544.042,Z 857.104,A -85,B 0,C 180,E1 23887.139,E2 23887.139} C_VEL
LIN {X 0,Y 541.371,Z 881.772,A -85,B 0,C 180,E1 23886.23,E2 23886.23} C_VEL
LIN {X 0,Y 538.764,Z 901.953,A -85,B 0,C 180,E1 23885.318,E2 23885.318} C_VEL
LIN {X 0,Y 535.739,Z 922.985,A -85,B 0,C 180,E1 23884.197,E2 23884.197} C_VEL
LIN {X 0,Y 533.867,Z 929.813,A -85,B 0,C 180,E1 23883.852,E2 23883.852} C_VEL
LIN {X 0,Y 526.058,Z 947.055,A -85,B 0,C 180,E1 23883.112,E2 23883.112} C_VEL
LIN {X 0,Y 524.043,Z 953.516,A -85,B 0,C 180,E1 23882.7,E2 23882.7} C_VEL
LIN {X 0,Y 520.487,Z 972.408,A -85,B 0,C 180,E1 23881.18,E2 23881.18} C_VEL
LIN {X 0,Y 516.696,Z 991.897,A -85,B 0,C 180,E1 23879.378,E2 23879.378} C_VEL
LIN {X 0,Y 513.126,Z 1009.24,A -85,B 0,C 180,E1 23877.505,E2 23877.505} C_VEL
LIN {X 0,Y 509.731,Z 1026.013,A -85,B 0,C 180,E1 23875.442,E2 23875.442} C_VEL
LIN {X 0,Y 506.602,Z 1041.262,A -85,B 0,C 180,E1 23873.25,E2 23873.25} C_VEL
LIN {X 0,Y 503.864,Z 1055.426,A -85,B 0,C 180,E1 23870.928,E2 23870.928} C_VEL
LIN {X 0,Y 501.496,Z 1068.148,A -85,B 0,C 180,E1 23868.483,E2 23868.483} C_VEL
LIN {X 0,Y 499.75,Z 1078.677,A -85,B 0,C 180,E1 23866.147,E2 23866.147} C_VEL
LIN {X 0,Y 498.183,Z 1089.338,A -85,B 0,C 180,E1 23863.345,E2 23863.345} C_VEL
LIN {X 0,Y 497.247,Z 1097.086,A -85,B 0,C 180,E1 23860.896,E2 23860.896} C_VEL
LIN {X 0,Y 496.531,Z 1104.554,A -85,B 0,C 180,E1 23857.987,E2 23857.987} C_VEL
LIN {X 0,Y 496.191,Z 1109.363,A -85,B 0,C 180,E1 23855.551,E2 23855.551} C_VEL
LIN {X 0,Y 496.025,Z 1113.152,A -85,B 0,C 180,E1 23853.004,E2 23853.004} C_VEL
LIN {X 0,Y 495.983,Z 1115.778,A -85,B 0,C 180,E1 23850.116,E2 23850.116} C_VEL
LIN {X 0,Y 495.94,Z 1116.727,A -85,B 0,C 180,E1 23847.689,E2 23847.689} C_VEL
LIN {X 0,Y 495.939,Z 1116.448,A -85,B 0,C 180,E1 23844.911,E2 23844.911} C_VEL
LIN {X 0,Y 495.993,Z 1114.592,A -85,B 0,C 180,E1 23842.237,E2 23842.237} C_VEL
LIN {X 0,Y 496.09,Z 1111.72,A -85,B 0,C 180,E1 23839.783,E2 23839.783} C_VEL
LIN {X 0,Y 496.378,Z 1106.652,A -85,B 0,C 180,E1 23836.843,E2 23836.843} C_VEL
LIN {X 0,Y 496.877,Z 1100.947,A -85,B 0,C 180,E1 23834.356,E2 23834.356} C_VEL
LIN {X 0,Y 497.768,Z 1093.202,A -85,B 0,C 180,E1 23831.617,E2 23831.617} C_VEL
LIN {X 0,Y 499.046,Z 1083.973,A -85,B 0,C 180,E1 23828.983,E2 23828.983} C_VEL
LIN {X 0,Y 500.867,Z 1073.138,A -85,B 0,C 180,E1 23826.343,E2 23826.343} C_VEL
LIN {X 0,Y 503.117,Z 1060.761,A -85,B 0,C 180,E1 23823.819,E2 23823.819} C_VEL
LIN {X 0,Y 505.845,Z 1047.275,A -85,B 0,C 180,E1 23821.422,E2 23821.422} C_VEL
LIN {X 0,Y 508.959,Z 1032.301,A -85,B 0,C 180,E1 23819.151,E2 23819.151} C_VEL
LIN {X 0,Y 512.233,Z 1017.154,A -85,B 0,C 180,E1 23817.135,E2 23817.135} C_VEL
LIN {X 0,Y 516.17,Z 998.679,A -85,B 0,C 180,E1 23815.013,E2 23815.013} C_VEL
LIN {X 0,Y 519.685,Z 982.056,A -85,B 0,C 180,E1 23813.353,E2 23813.353} C_VEL
LIN {X 0,Y 523.972,Z 960.868,A -85,B 0,C 180,E1 23811.53,E2 23811.53} C_VEL
LIN {X 0,Y 527.348,Z 943.079,A -85,B 0,C 180,E1 23810.214,E2 23810.214} C_VEL
LIN {X 0,Y 531.068,Z 921.98,A -85,B 0,C 180,E1 23808.862,E2 23808.862} C_VEL
LIN {X 0,Y 534.39,Z 900.726,A -85,B 0,C 180,E1 23807.727,E2 23807.727} C_VEL
LIN {X 0,Y 537.505,Z 878.445,A -85,B 0,C 180,E1 23806.725,E2 23806.725} C_VEL
LIN {X 0,Y 540.19,Z 854.693,A -85,B 0,C 180,E1 23805.876,E2 23805.876} C_VEL
LIN {X 0,Y 542.362,Z 831.672,A -85,B 0,C 180,E1 23805.231,E2 23805.231} C_VEL
LIN {X 0,Y 543.966,Z 806.948,A -85,B 0,C 180,E1 23804.732,E2 23804.732} C_VEL
LIN {X 0,Y 552.32,Z 575.484,A -85,B 0,C 180,E1 23801.354,E2 23801.354} C_VEL
LIN {X 0,Y 554.744,Z 508.095,A -85,B 0,C 180,E1 23800.359,E2 23800.359} C_VEL
LIN {X 0,Y 541.272,Z 487.786,A -85,B 0,C 180,E1 23798.333,E2 23798.333} C_VEL
LIN {X 0,Y 527.634,Z 468.88,A -85,B 0,C 180,E1 23796.112,E2 23796.112} C_VEL
LIN {X 0,Y 519.136,Z 457.855,A -85,B 0,C 180,E1 23794.624,E2 23794.624} C_VEL
LIN {X 0,Y 515,Z 452.554,A -85,B 0,C 180,E1 23793.864,E2 23793.864} C_VEL
LIN {X 0,Y 511.063,Z 447.608,A -85,B 0,C 180,E1 23793.117,E2 23793.117} C_VEL
LIN {X 0,Y 507.824,Z 443.561,A -85,B 0,C 180,E1 23792.482,E2 23792.482} C_VEL
LIN {X 0,Y 506.724,Z 442.099,A -85,B 0,C 180,E1 23792.26,E2 23792.26} C_VEL
LIN {X 0,Y 503.753,Z 438.918,A -85,B 0,C 180,E1 23791.669,E2 23791.669} C_VEL
LIN {X 0,Y 502.406,Z 436.455,A -85,B 0,C 180,E1 23791.369,E2 23791.369} C_VEL
LIN {X 0,Y 499.427,Z 433.88,A -85,B 0,C 180,E1 23790.766,E2 23790.766} C_VEL
LIN {X 0,Y 498.053,Z 431.061,A -85,B 0,C 180,E1 23790.392,E2 23790.392} C_VEL
LIN {X 0,Y 497.867,Z 430.202,A -85,B 0,C 180,E1 23790.005,E2 23790.005} C_VEL
LIN {X 0,Y 497.92,Z 430.184,A -85,B 0,C 180,E1 23786.668,E2 23786.668} C_VEL
LIN {X 0,Y 497.893,Z 430.192,A -85,B 0,C 180,E1 23783.18,E2 23783.18} C_VEL
LIN {X 0,Y 497.877,Z 430.185,A -85,B 0,C 180,E1 23779.718,E2 23779.718} C_VEL
LIN {X 0,Y 497.913,Z 430.178,A -85,B 0,C 180,E1 23776.279,E2 23776.279} C_VEL
LIN {X 0,Y 497.917,Z 430.197,A -85,B 0,C 180,E1 23772.88,E2 23772.88} C_VEL
LIN {X 0,Y 497.892,Z 430.21,A -85,B 0,C 180,E1 23769.362,E2 23769.362} C_VEL
LIN {X 0,Y 497.9,Z 430.186,A -85,B 0,C 180,E1 23765.763,E2 23765.763} C_VEL
LIN {X 0,Y 497.926,Z 430.171,A -85,B 0,C 180,E1 23762.302,E2 23762.302} C_VEL
LIN {X 0,Y 497.923,Z 430.19,A -85,B 0,C 180,E1 23758.734,E2 23758.734} C_VEL
LIN {X 0,Y 497.908,Z 430.202,A -85,B 0,C 180,E1 23755.162,E2 23755.162} C_VEL
LIN {X 0,Y 497.916,Z 430.18,A -85,B 0,C 180,E1 23751.57,E2 23751.57} C_VEL
LIN {X 0,Y 497.922,Z 430.174,A -85,B 0,C 180,E1 23748.063,E2 23748.063} C_VEL
LIN {X 0,Y 497.929,Z 430.191,A -85,B 0,C 180,E1 23744.51,E2 23744.51} C_VEL
LIN {X 0,Y 497.924,Z 430.21,A -85,B 0,C 180,E1 23740.894,E2 23740.894} C_VEL
LIN {X 0,Y 497.927,Z 430.167,A -85,B 0,C 180,E1 23737.322,E2 23737.322} C_VEL
LIN {X 0,Y 497.911,Z 430.167,A -85,B 0,C 180,E1 23733.852,E2 23733.852} C_VEL
LIN {X 0,Y 497.916,Z 430.193,A -85,B 0,C 180,E1 23730.263,E2 23730.263} C_VEL
LIN {X 0,Y 497.962,Z 430.42,A -85,B 0,C 180,E1 23728.697,E2 23728.697} C_VEL
LIN {X 0,Y 499.412,Z 433.945,A -85,B 0,C 180,E1 23727.821,E2 23727.821} C_VEL
LIN {X 0,Y 500.602,Z 436.381,A -85,B 0,C 180,E1 23727.228,E2 23727.228} C_VEL
LIN {X 0,Y 502.629,Z 440.464,A -85,B 0,C 180,E1 23726.257,E2 23726.257} C_VEL
LIN {X 0,Y 504.349,Z 443.514,A -85,B 0,C 180,E1 23725.596,E2 23725.596} C_VEL
LIN {X 0,Y 516.109,Z 459.712,A -85,B 0,C 180,E1 23723.261,E2 23723.261} C_VEL
LIN {X 0,Y 525.438,Z 472.996,A -85,B 0,C 180,E1 23721.57,E2 23721.57} C_VEL
LIN {X 0,Y 536.768,Z 490.223,A -85,B 0,C 180,E1 23719.66,E2 23719.66} C_VEL
LIN {X 0,Y 547.858,Z 508.268,A -85,B 0,C 180,E1 23717.912,E2 23717.912} C_VEL
LIN {X 0,Y 554.675,Z 520.539,A -85,B 0,C 180,E1 23716.879,E2 23716.879} C_VEL
LIN {X 0,Y 546.591,Z 745.359,A -85,B 0,C 180,E1 23713.601,E2 23713.601} C_VEL
LIN {X 0,Y 543.241,Z 838.498,A -85,B 0,C 180,E1 23712.228,E2 23712.228} C_VEL
LIN {X 0,Y 541.271,Z 864.297,A -85,B 0,C 180,E1 23711.69,E2 23711.69} C_VEL
LIN {X 0,Y 539.136,Z 885.058,A -85,B 0,C 180,E1 23711.111,E2 23711.111} C_VEL
LIN {X 0,Y 536.349,Z 907.913,A -85,B 0,C 180,E1 23710.308,E2 23710.308} C_VEL
LIN {X 0,Y 533.167,Z 929.931,A -85,B 0,C 180,E1 23709.337,E2 23709.337} C_VEL
LIN {X 0,Y 529.656,Z 951.855,A -85,B 0,C 180,E1 23708.189,E2 23708.189} C_VEL
LIN {X 0,Y 525.752,Z 973.735,A -85,B 0,C 180,E1 23706.804,E2 23706.804} C_VEL
LIN {X 0,Y 522.014,Z 993.606,A -85,B 0,C 180,E1 23705.343,E2 23705.343} C_VEL
LIN {X 0,Y 517.931,Z 1014.053,A -85,B 0,C 180,E1 23703.578,E2 23703.578} C_VEL
LIN {X 0,Y 514.491,Z 1030.893,A -85,B 0,C 180,E1 23701.912,E2 23701.912} C_VEL
LIN {X 0,Y 510.504,Z 1050.223,A -85,B 0,C 180,E1 23699.705,E2 23699.705} C_VEL
LIN {X 0,Y 507.459,Z 1065.378,A -85,B 0,C 180,E1 23697.711,E2 23697.711} C_VEL
LIN {X 0,Y 504.285,Z 1081.765,A -85,B 0,C 180,E1 23695.233,E2 23695.233} C_VEL
LIN {X 0,Y 501.96,Z 1094.639,A -85,B 0,C 180,E1 23692.981,E2 23692.981} C_VEL
LIN {X 0,Y 499.769,Z 1108.137,A -85,B 0,C 180,E1 23690.25,E2 23690.25} C_VEL
LIN {X 0,Y 498.356,Z 1118.12,A -85,B 0,C 180,E1 23687.877,E2 23687.877} C_VEL
LIN {X 0,Y 497.232,Z 1127.953,A -85,B 0,C 180,E1 23685.15,E2 23685.15} C_VEL
LIN {X 0,Y 496.547,Z 1135.515,A -85,B 0,C 180,E1 23682.561,E2 23682.561} C_VEL
LIN {X 0,Y 496.172,Z 1141.424,A -85,B 0,C 180,E1 23680.098,E2 23680.098} C_VEL
LIN {X 0,Y 495.982,Z 1146.709,A -85,B 0,C 180,E1 23677.18,E2 23677.18} C_VEL
LIN {X 0,Y 495.932,Z 1149.611,A -85,B 0,C 180,E1 23674.858,E2 23674.858} C_VEL
LIN {X 0,Y 495.928,Z 1151.414,A -85,B 0,C 180,E1 23672.542,E2 23672.542} C_VEL
LIN {X 0,Y 495.935,Z 1152.124,A -85,B 0,C 180,E1 23669.769,E2 23669.769} C_VEL
LIN {X 0,Y 495.923,Z 1151.34,A -85,B 0,C 180,E1 23667.342,E2 23667.342} C_VEL
LIN {X 0,Y 495.932,Z 1149.603,A -85,B 0,C 180,E1 23665.142,E2 23665.142} C_VEL
LIN {X 0,Y 495.978,Z 1146.511,A -85,B 0,C 180,E1 23662.692,E2 23662.692} C_VEL
LIN {X 0,Y 496.171,Z 1141.371,A -85,B 0,C 180,E1 23659.902,E2 23659.902} C_VEL
LIN {X 0,Y 496.545,Z 1135.424,A -85,B 0,C 180,E1 23657.439,E2 23657.439} C_VEL
LIN {X 0,Y 497.265,Z 1127.382,A -85,B 0,C 180,E1 23654.727,E2 23654.727} C_VEL
LIN {X 0,Y 498.337,Z 1117.85,A -85,B 0,C 180,E1 23652.122,E2 23652.122} C_VEL
LIN {X 0,Y 499.897,Z 1106.697,A -85,B 0,C 180,E1 23649.511,E2 23649.511} C_VEL
LIN {X 0,Y 501.929,Z 1093.805,A -85,B 0,C 180,E1 23646.978,E2 23646.978} C_VEL
LIN {X 0,Y 504.321,Z 1080.214,A -85,B 0,C 180,E1 23644.643,E2 23644.643} C_VEL
LIN {X 0,Y 507.135,Z 1065.012,A -85,B 0,C 180,E1 23642.397,E2 23642.397} C_VEL
LIN {X 0,Y 510.007,Z 1050.096,A -85,B 0,C 180,E1 23640.457,E2 23640.457} C_VEL
LIN {X 0,Y 513.842,Z 1030.547,A -85,B 0,C 180,E1 23638.252,E2 23638.252} C_VEL
LIN {X 0,Y 517.064,Z 1013.966,A -85,B 0,C 180,E1 23636.628,E2 23636.628} C_VEL
LIN {X 0,Y 521.037,Z 992.937,A -85,B 0,C 180,E1 23634.837,E2 23634.837} C_VEL
LIN {X 0,Y 524.481,Z 973.665,A -85,B 0,C 180,E1 23633.433,E2 23633.433} C_VEL
LIN {X 0,Y 528.119,Z 952.119,A -85,B 0,C 180,E1 23632.076,E2 23632.076} C_VEL
LIN {X 0,Y 531.454,Z 930.13,A -85,B 0,C 180,E1 23630.929,E2 23630.929} C_VEL
LIN {X 0,Y 534.611,Z 907.091,A -85,B 0,C 180,E1 23629.92,E2 23629.92} C_VEL
LIN {X 0,Y 537.247,Z 883.92,A -85,B 0,C 180,E1 23629.119,E2 23629.119} C_VEL
LIN {X 0,Y 539.318,Z 862.502,A -85,B 0,C 180,E1 23628.533,E2 23628.533} C_VEL
LIN {X 0,Y 541.099,Z 836.356,A -85,B 0,C 180,E1 23628.007,E2 23628.007} C_VEL
LIN {X 0,Y 548.366,Z 613.389,A -85,B 0,C 180,E1 23624.782,E2 23624.782} C_VEL
LIN {X 0,Y 551.409,Z 518.621,A -85,B 0,C 180,E1 23623.396,E2 23623.396} C_VEL
LIN {X 0,Y 538.009,Z 495.343,A -85,B 0,C 180,E1 23621.498,E2 23621.498} C_VEL
LIN {X 0,Y 525.007,Z 474.383,A -85,B 0,C 180,E1 23619.526,E2 23619.526} C_VEL
LIN {X 0,Y 512.211,Z 455.572,A -85,B 0,C 180,E1 23617.451,E2 23617.451} C_VEL
LIN {X 0,Y 503.976,Z 443.621,A -85,B 0,C 180,E1 23615.963,E2 23615.963} C_VEL
LIN {X 0,Y 500.844,Z 437.21,A -85,B 0,C 180,E1 23614.662,E2 23614.662} C_VEL
LIN {X 0,Y 499.332,Z 433.854,A -85,B 0,C 180,E1 23613.965,E2 23613.965} C_VEL
LIN {X 0,Y 497.948,Z 430.32,A -85,B 0,C 180,E1 23613.174,E2 23613.174} C_VEL
LIN {X 0,Y 497.921,Z 430.179,A -85,B 0,C 180,E1 23609.596,E2 23609.596} C_VEL
LIN {X 0,Y 497.915,Z 430.205,A -85,B 0,C 180,E1 23606.09,E2 23606.09} C_VEL
LIN {X 0,Y 497.934,Z 430.188,A -85,B 0,C 180,E1 23602.524,E2 23602.524} C_VEL
LIN {X 0,Y 497.918,Z 430.172,A -85,B 0,C 180,E1 23598.943,E2 23598.943} C_VEL
LIN {X 0,Y 497.93,Z 430.184,A -85,B 0,C 180,E1 23595.371,E2 23595.371} C_VEL
LIN {X 0,Y 497.924,Z 430.204,A -85,B 0,C 180,E1 23591.819,E2 23591.819} C_VEL
LIN {X 0,Y 497.925,Z 430.168,A -85,B 0,C 180,E1 23588.197,E2 23588.197} C_VEL
LIN {X 0,Y 497.906,Z 430.192,A -85,B 0,C 180,E1 23584.723,E2 23584.723} C_VEL
LIN {X 0,Y 497.921,Z 430.197,A -85,B 0,C 180,E1 23581.151,E2 23581.151} C_VEL
LIN {X 0,Y 497.925,Z 430.166,A -85,B 0,C 180,E1 23577.583,E2 23577.583} C_VEL
LIN {X 0,Y 497.918,Z 430.204,A -85,B 0,C 180,E1 23574.006,E2 23574.006} C_VEL
LIN {X 0,Y 497.89,Z 430.185,A -85,B 0,C 180,E1 23570.521,E2 23570.521} C_VEL
LIN {X 0,Y 497.908,Z 430.172,A -85,B 0,C 180,E1 23567.002,E2 23567.002} C_VEL
LIN {X 0,Y 497.929,Z 430.208,A -85,B 0,C 180,E1 23563.552,E2 23563.552} C_VEL
LIN {X 0,Y 497.885,Z 430.183,A -85,B 0,C 180,E1 23560.031,E2 23560.031} C_VEL
LIN {X 0,Y 497.874,Z 430.175,A -85,B 0,C 180,E1 23556.443,E2 23556.443} C_VEL
LIN {X 0,Y 497.916,Z 430.198,A -85,B 0,C 180,E1 23553.009,E2 23553.009} C_VEL
LIN {X 0,Y 497.892,Z 430.208,A -85,B 0,C 180,E1 23549.597,E2 23549.597} C_VEL
LIN {X 0,Y 497.86,Z 430.192,A -85,B 0,C 180,E1 23546.198,E2 23546.198} C_VEL
LIN {X 0,Y 497.894,Z 430.184,A -85,B 0,C 180,E1 23542.808,E2 23542.808} C_VEL
LIN {X 0,Y 497.881,Z 430.377,A -85,B 0,C 180,E1 23541.862,E2 23541.862} C_VEL
LIN {X 0,Y 498.262,Z 431.875,A -85,B 0,C 180,E1 23541.604,E2 23541.604} C_VEL
LIN {X 0,Y 500.182,Z 434.872,A -85,B 0,C 180,E1 23541.231,E2 23541.231} C_VEL
LIN {X 0,Y 502.271,Z 436.71,A -85,B 0,C 180,E1 23540.871,E2 23540.871} C_VEL
LIN {X 0,Y 504.79,Z 440.552,A -85,B 0,C 180,E1 23540.407,E2 23540.407} C_VEL
LIN {X 0,Y 506.88,Z 442.757,A -85,B 0,C 180,E1 23540.052,E2 23540.052} C_VEL
LIN {X 0,Y 510.339,Z 447.136,A -85,B 0,C 180,E1 23539.459,E2 23539.459} C_VEL
LIN {X 0,Y 514.393,Z 452.512,A -85,B 0,C 180,E1 23538.779,E2 23538.779} C_VEL
LIN {X 0,Y 529.161,Z 472.835,A -85,B 0,C 180,E1 23536.45,E2 23536.45} C_VEL
LIN {X 0,Y 542.262,Z 492.076,A -85,B 0,C 180,E1 23534.547,E2 23534.547} C_VEL
LIN {X 0,Y 551.746,Z 507.102,A -85,B 0,C 180,E1 23533.241,E2 23533.241} C_VEL
LIN {X 0,Y 543.581,Z 751.145,A -85,B 0,C 180,E1 23529.725,E2 23529.725} C_VEL
LIN {X 0,Y 541.468,Z 811.428,A -85,B 0,C 180,E1 23528.833,E2 23528.833} C_VEL
LIN {X 0,Y 539.786,Z 835.931,A -85,B 0,C 180,E1 23528.297,E2 23528.297} C_VEL
LIN {X 0,Y 537.826,Z 857.475,A -85,B 0,C 180,E1 23527.674,E2 23527.674} C_VEL
LIN {X 0,Y 535.143,Z 881.467,A -85,B 0,C 180,E1 23526.787,E2 23526.787} C_VEL
LIN {X 0,Y 532.443,Z 901.723,A -85,B 0,C 180,E1 23525.868,E2 23525.868} C_VEL
LIN {X 0,Y 529.113,Z 923.998,A -85,B 0,C 180,E1 23524.668,E2 23524.668} C_VEL
LIN {X 0,Y 525.659,Z 944.41,A -85,B 0,C 180,E1 23523.348,E2 23523.348} C_VEL
LIN {X 0,Y 524.043,Z 953.516,A -85,B 0,C 180,E1 23522.7,E2 23522.7} C_VEL
LIN {X 0,Y 522.018,Z 959.959,A -85,B 0,C 180,E1 23522.268,E2 23522.268} C_VEL
LIN {X 0,Y 513.5,Z 977.068,A -85,B 0,C 180,E1 23521.248,E2 23521.248} C_VEL
LIN {X 0,Y 511.785,Z 982.184,A -85,B 0,C 180,E1 23520.821,E2 23520.821} C_VEL
LIN {X 0,Y 508.276,Z 998.992,A -85,B 0,C 180,E1 23519.138,E2 23519.138} C_VEL
LIN {X 0,Y 504.354,Z 1017.515,A -85,B 0,C 180,E1 23517.001,E2 23517.001} C_VEL
LIN {X 0,Y 501.164,Z 1032.327,A -85,B 0,C 180,E1 23515.022,E2 23515.022} C_VEL
LIN {X 0,Y 497.96,Z 1047.715,A -85,B 0,C 180,E1 23512.677,E2 23512.677} C_VEL
LIN {X 0,Y 495.287,Z 1060.918,A -85,B 0,C 180,E1 23510.318,E2 23510.318} C_VEL
LIN {X 0,Y 493.039,Z 1073.071,A -85,B 0,C 180,E1 23507.832,E2 23507.832} C_VEL
LIN {X 0,Y 491.208,Z 1083.773,A -85,B 0,C 180,E1 23505.224,E2 23505.224} C_VEL
LIN {X 0,Y 489.944,Z 1092.505,A -85,B 0,C 180,E1 23502.733,E2 23502.733} C_VEL
LIN {X 0,Y 488.963,Z 1100.679,A -85,B 0,C 180,E1 23499.891,E2 23499.891} C_VEL
LIN {X 0,Y 488.453,Z 1106.155,A -85,B 0,C 180,E1 23497.528,E2 23497.528} C_VEL
LIN {X 0,Y 488.145,Z 1111.121,A -85,B 0,C 180,E1 23494.818,E2 23494.818} C_VEL
LIN {X 0,Y 488.005,Z 1114.585,A -85,B 0,C 180,E1 23491.996,E2 23491.996} C_VEL
LIN {X 0,Y 487.966,Z 1116.418,A -85,B 0,C 180,E1 23489.53,E2 23489.53} C_VEL
LIN {X 0,Y 487.94,Z 1117.094,A -85,B 0,C 180,E1 23486.593,E2 23486.593} C_VEL
LIN {X 0,Y 487.969,Z 1116.245,A -85,B 0,C 180,E1 23484.001,E2 23484.001} C_VEL
LIN {X 0,Y 488.036,Z 1114.066,A -85,B 0,C 180,E1 23481.28,E2 23481.28} C_VEL
LIN {X 0,Y 488.211,Z 1110.122,A -85,B 0,C 180,E1 23478.421,E2 23478.421} C_VEL
LIN {X 0,Y 488.566,Z 1105.362,A -85,B 0,C 180,E1 23475.904,E2 23475.904} C_VEL
LIN {X 0,Y 489.345,Z 1097.968,A -85,B 0,C 180,E1 23472.888,E2 23472.888} C_VEL
LIN {X 0,Y 490.381,Z 1090.166,A -85,B 0,C 180,E1 23470.34,E2 23470.34} C_VEL
LIN {X 0,Y 492.042,Z 1079.926,A -85,B 0,C 180,E1 23467.54,E2 23467.54} C_VEL
LIN {X 0,Y 494.091,Z 1068.712,A -85,B 0,C 180,E1 23464.979,E2 23464.979} C_VEL
LIN {X 0,Y 496.742,Z 1055.739,A -85,B 0,C 180,E1 23462.421,E2 23462.421} C_VEL
LIN {X 0,Y 499.673,Z 1042.009,A -85,B 0,C 180,E1 23460.114,E2 23460.114} C_VEL
LIN {X 0,Y 503.182,Z 1026.439,A -85,B 0,C 180,E1 23457.822,E2 23457.822} C_VEL
LIN {X 0,Y 506.878,Z 1009.918,A -85,B 0,C 180,E1 23455.745,E2 23455.745} C_VEL
LIN {X 0,Y 510.665,Z 993.106,A -85,B 0,C 180,E1 23453.888,E2 23453.888} C_VEL
LIN {X 0,Y 514.814,Z 973.76,A -85,B 0,C 180,E1 23452.05,E2 23452.05} C_VEL
LIN {X 0,Y 518.566,Z 955.595,A -85,B 0,C 180,E1 23450.555,E2 23450.555} C_VEL
LIN {X 0,Y 522.792,Z 933.53,A -85,B 0,C 180,E1 23449.003,E2 23449.003} C_VEL
LIN {X 0,Y 526.1,Z 914.479,A -85,B 0,C 180,E1 23447.863,E2 23447.863} C_VEL
LIN {X 0,Y 529.633,Z 892.307,A -85,B 0,C 180,E1 23446.74,E2 23446.74} C_VEL
LIN {X 0,Y 532.498,Z 870.595,A -85,B 0,C 180,E1 23445.842,E2 23445.842} C_VEL
LIN {X 0,Y 535.062,Z 848.092,A -85,B 0,C 180,E1 23445.084,E2 23445.084} C_VEL
LIN {X 0,Y 537.142,Z 823.966,A -85,B 0,C 180,E1 23444.472,E2 23444.472} C_VEL
LIN {X 0,Y 538.437,Z 802.227,A -85,B 0,C 180,E1 23444.065,E2 23444.065} C_VEL
LIN {X 0,Y 547.812,Z 551.543,A -85,B 0,C 180,E1 23440.387,E2 23440.387} C_VEL
LIN {X 0,Y 549.231,Z 511.767,A -85,B 0,C 180,E1 23439.786,E2 23439.786} C_VEL
LIN {X 0,Y 536.642,Z 492.823,A -85,B 0,C 180,E1 23437.841,E2 23437.841} C_VEL
LIN {X 0,Y 524.11,Z 475.274,A -85,B 0,C 180,E1 23435.751,E2 23435.751} C_VEL
LIN {X 0,Y 515.698,Z 464.267,A -85,B 0,C 180,E1 23434.248,E2 23434.248} C_VEL
LIN {X 0,Y 511.348,Z 458.703,A -85,B 0,C 180,E1 23433.431,E2 23433.431} C_VEL
LIN {X 0,Y 507.838,Z 454.254,A -85,B 0,C 180,E1 23432.749,E2 23432.749} C_VEL
LIN {X 0,Y 504.291,Z 449.539,A -85,B 0,C 180,E1 23432.032,E2 23432.032} C_VEL
LIN {X 0,Y 500.621,Z 445.472,A -85,B 0,C 180,E1 23431.285,E2 23431.285} C_VEL
LIN {X 0,Y 499.233,Z 443.322,A -85,B 0,C 180,E1 23430.98,E2 23430.98} C_VEL
LIN {X 0,Y 496.12,Z 440.109,A -85,B 0,C 180,E1 23430.322,E2 23430.322} C_VEL
LIN {X 0,Y 494.566,Z 437.479,A -85,B 0,C 180,E1 23429.959,E2 23429.959} C_VEL
LIN {X 0,Y 491.486,Z 434.924,A -85,B 0,C 180,E1 23429.293,E2 23429.293} C_VEL
LIN {X 0,Y 490.163,Z 432.096,A -85,B 0,C 180,E1 23428.912,E2 23428.912} C_VEL
LIN {X 0,Y 489.972,Z 431.204,A -85,B 0,C 180,E1 23428.524,E2 23428.524} C_VEL
LIN {X 0,Y 489.97,Z 431.176,A -85,B 0,C 180,E1 23424.988,E2 23424.988} C_VEL
LIN {X 0,Y 489.936,Z 431.191,A -85,B 0,C 180,E1 23421.553,E2 23421.553} C_VEL
LIN {X 0,Y 489.952,Z 431.202,A -85,B 0,C 180,E1 23417.948,E2 23417.948} C_VEL
LIN {X 0,Y 489.995,Z 431.18,A -85,B 0,C 180,E1 23414.416,E2 23414.416} C_VEL
LIN {X 0,Y 489.979,Z 431.167,A -85,B 0,C 180,E1 23410.821,E2 23410.821} C_VEL
LIN {X 0,Y 489.951,Z 431.17,A -85,B 0,C 180,E1 23407.328,E2 23407.328} C_VEL
LIN {X 0,Y 489.962,Z 431.189,A -85,B 0,C 180,E1 23403.686,E2 23403.686} C_VEL
LIN {X 0,Y 489.998,Z 431.185,A -85,B 0,C 180,E1 23400.117,E2 23400.117} C_VEL
LIN {X 0,Y 489.984,Z 431.161,A -85,B 0,C 180,E1 23396.49,E2 23396.49} C_VEL
LIN {X 0,Y 489.973,Z 431.163,A -85,B 0,C 180,E1 23392.967,E2 23392.967} C_VEL
LIN {X 0,Y 489.976,Z 431.187,A -85,B 0,C 180,E1 23389.417,E2 23389.417} C_VEL
LIN {X 0,Y 489.995,Z 431.196,A -85,B 0,C 180,E1 23385.765,E2 23385.765} C_VEL
LIN {X 0,Y 489.981,Z 431.174,A -85,B 0,C 180,E1 23382.176,E2 23382.176} C_VEL
LIN {X 0,Y 489.988,Z 431.146,A -85,B 0,C 180,E1 23378.575,E2 23378.575} C_VEL
LIN {X 0,Y 489.986,Z 431.178,A -85,B 0,C 180,E1 23374.966,E2 23374.966} C_VEL
LIN {X 0,Y 489.995,Z 431.181,A -85,B 0,C 180,E1 23371.339,E2 23371.339} C_VEL
LIN {X 0,Y 490.027,Z 431.56,A -85,B 0,C 180,E1 23370.031,E2 23370.031} C_VEL
LIN {X 0,Y 491.487,Z 434.912,A -85,B 0,C 180,E1 23369.152,E2 23369.152} C_VEL
LIN {X 0,Y 492.458,Z 436.636,A -85,B 0,C 180,E1 23368.682,E2 23368.682} C_VEL
LIN {X 0,Y 495.108,Z 442.241,A -85,B 0,C 180,E1 23367.309,E2 23367.309} C_VEL
LIN {X 0,Y 502.465,Z 452.07,A -85,B 0,C 180,E1 23365.691,E2 23365.691} C_VEL
LIN {X 0,Y 511.852,Z 464.733,A -85,B 0,C 180,E1 23363.812,E2 23363.812} C_VEL
LIN {X 0,Y 524.794,Z 483.65,A -85,B 0,C 180,E1 23361.427,E2 23361.427} C_VEL
LIN {X 0,Y 536.954,Z 502.694,A -85,B 0,C 180,E1 23359.379,E2 23359.379} C_VEL
LIN {X 0,Y 548.47,Z 522.397,A -85,B 0,C 180,E1 23357.564,E2 23357.564} C_VEL
LIN {X 0,Y 549.179,Z 524.132,A -85,B 0,C 180,E1 23357.447,E2 23357.447} C_VEL
LIN {X 0,Y 540.818,Z 747.848,A -85,B 0,C 180,E1 23354.16,E2 23354.16} C_VEL
LIN {X 0,Y 537.427,Z 838.283,A -85,B 0,C 180,E1 23352.816,E2 23352.816} C_VEL
LIN {X 0,Y 535.393,Z 864.063,A -85,B 0,C 180,E1 23352.275,E2 23352.275} C_VEL
LIN {X 0,Y 533.199,Z 884.694,A -85,B 0,C 180,E1 23351.697,E2 23351.697} C_VEL
LIN {X 0,Y 530.238,Z 908.046,A -85,B 0,C 180,E1 23350.871,E2 23350.871} C_VEL
LIN {X 0,Y 527.143,Z 928.771,A -85,B 0,C 180,E1 23349.954,E2 23349.954} C_VEL
LIN {X 0,Y 523.812,Z 948.88,A -85,B 0,C 180,E1 23348.904,E2 23348.904} C_VEL
LIN {X 0,Y 519.563,Z 972.081,A -85,B 0,C 180,E1 23347.455,E2 23347.455} C_VEL
LIN {X 0,Y 515.853,Z 990.957,A -85,B 0,C 180,E1 23346.071,E2 23346.071} C_VEL
LIN {X 0,Y 511.328,Z 1012.869,A -85,B 0,C 180,E1 23344.191,E2 23344.191} C_VEL
LIN {X 0,Y 507.744,Z 1029.656,A -85,B 0,C 180,E1 23342.522,E2 23342.522} C_VEL
LIN {X 0,Y 503.748,Z 1048.203,A -85,B 0,C 180,E1 23340.408,E2 23340.408} C_VEL
LIN {X 0,Y 500.481,Z 1063.504,A -85,B 0,C 180,E1 23338.391,E2 23338.391} C_VEL
LIN {X 0,Y 497.39,Z 1078.721,A -85,B 0,C 180,E1 23336.12,E2 23336.12} C_VEL
LIN {X 0,Y 494.664,Z 1092.61,A -85,B 0,C 180,E1 23333.698,E2 23333.698} C_VEL
LIN {X 0,Y 492.532,Z 1104.758,A -85,B 0,C 180,E1 23331.279,E2 23331.279} C_VEL
LIN {X 0,Y 490.722,Z 1116.484,A -85,B 0,C 180,E1 23328.534,E2 23328.534} C_VEL
LIN {X 0,Y 489.587,Z 1125.258,A -85,B 0,C 180,E1 23326.126,E2 23326.126} C_VEL
LIN {X 0,Y 488.671,Z 1134.329,A -85,B 0,C 180,E1 23323.128,E2 23323.128} C_VEL
LIN {X 0,Y 488.234,Z 1140.381,A -85,B 0,C 180,E1 23320.621,E2 23320.621} C_VEL
LIN {X 0,Y 487.996,Z 1145.592,A -85,B 0,C 180,E1 23317.891,E2 23317.891} C_VEL
LIN {X 0,Y 487.927,Z 1149.114,A -85,B 0,C 180,E1 23315.161,E2 23315.161} C_VEL
LIN {X 0,Y 487.924,Z 1150.995,A -85,B 0,C 180,E1 23312.819,E2 23312.819} C_VEL
LIN {X 0,Y 487.94,Z 1151.845,A -85,B 0,C 180,E1 23310.235,E2 23310.235} C_VEL
LIN {X 0,Y 487.93,Z 1151.119,A -85,B 0,C 180,E1 23307.416,E2 23307.416} C_VEL
LIN {X 0,Y 487.933,Z 1149.307,A -85,B 0,C 180,E1 23305.063,E2 23305.063} C_VEL
LIN {X 0,Y 487.977,Z 1146.225,A -85,B 0,C 180,E1 23302.583,E2 23302.583} C_VEL
LIN {X 0,Y 488.188,Z 1141.057,A -85,B 0,C 180,E1 23299.736,E2 23299.736} C_VEL
LIN {X 0,Y 488.587,Z 1135.101,A -85,B 0,C 180,E1 23297.231,E2 23297.231} C_VEL
LIN {X 0,Y 489.354,Z 1127.043,A -85,B 0,C 180,E1 23294.474,E2 23294.474} C_VEL
LIN {X 0,Y 490.494,Z 1117.5,A -85,B 0,C 180,E1 23291.826,E2 23291.826} C_VEL
LIN {X 0,Y 492.148,Z 1106.277,A -85,B 0,C 180,E1 23289.16,E2 23289.16} C_VEL
LIN {X 0,Y 494.251,Z 1093.629,A -85,B 0,C 180,E1 23286.639,E2 23286.639} C_VEL
LIN {X 0,Y 496.815,Z 1079.818,A -85,B 0,C 180,E1 23284.232,E2 23284.232} C_VEL
LIN {X 0,Y 499.837,Z 1064.256,A -85,B 0,C 180,E1 23281.908,E2 23281.908} C_VEL
LIN {X 0,Y 502.877,Z 1049.188,A -85,B 0,C 180,E1 23279.93,E2 23279.93} C_VEL
LIN {X 0,Y 506.819,Z 1029.975,A -85,B 0,C 180,E1 23277.747,E2 23277.747} C_VEL
LIN {X 0,Y 510.204,Z 1013.268,A -85,B 0,C 180,E1 23276.096,E2 23276.096} C_VEL
LIN {X 0,Y 514.413,Z 991.763,A -85,B 0,C 180,E1 23274.256,E2 23274.256} C_VEL
LIN {X 0,Y 517.915,Z 972.935,A -85,B 0,C 180,E1 23272.877,E2 23272.877} C_VEL
LIN {X 0,Y 521.789,Z 950.738,A -85,B 0,C 180,E1 23271.48,E2 23271.48} C_VEL
LIN {X 0,Y 525.132,Z 929.47,A -85,B 0,C 180,E1 23270.367,E2 23270.367} C_VEL
LIN {X 0,Y 528.352,Z 906.743,A -85,B 0,C 180,E1 23269.366,E2 23269.366} C_VEL
LIN {X 0,Y 531.073,Z 883.605,A -85,B 0,C 180,E1 23268.563,E2 23268.563} C_VEL
LIN {X 0,Y 533.195,Z 862.36,A -85,B 0,C 180,E1 23267.978,E2 23267.978} C_VEL
LIN {X 0,Y 535.039,Z 836.15,A -85,B 0,C 180,E1 23267.446,E2 23267.446} C_VEL
LIN {X 0,Y 542.588,Z 613.761,A -85,B 0,C 180,E1 23264.202,E2 23264.202} C_VEL
LIN {X 0,Y 545.655,Z 522.019,A -85,B 0,C 180,E1 23262.848,E2 23262.848} C_VEL
LIN {X 0,Y 533.295,Z 500.33,A -85,B 0,C 180,E1 23261.049,E2 23261.049} C_VEL
LIN {X 0,Y 520.834,Z 480.13,A -85,B 0,C 180,E1 23259.116,E2 23259.116} C_VEL
LIN {X 0,Y 508.468,Z 461.76,A -85,B 0,C 180,E1 23257.066,E2 23257.066} C_VEL
LIN {X 0,Y 498.776,Z 448.147,A -85,B 0,C 180,E1 23255.335,E2 23255.335} C_VEL
LIN {X 0,Y 495.504,Z 443.368,A -85,B 0,C 180,E1 23254.685,E2 23254.685} C_VEL
LIN {X 0,Y 491.536,Z 434.993,A -85,B 0,C 180,E1 23252.898,E2 23252.898} C_VEL
LIN {X 0,Y 489.984,Z 431.299,A -85,B 0,C 180,E1 23252.027,E2 23252.027} C_VEL
LIN {X 0,Y 489.981,Z 431.161,A -85,B 0,C 180,E1 23248.391,E2 23248.391} C_VEL
LIN {X 0,Y 489.985,Z 431.161,A -85,B 0,C 180,E1 23244.858,E2 23244.858} C_VEL
LIN {X 0,Y 489.992,Z 431.195,A -85,B 0,C 180,E1 23241.299,E2 23241.299} C_VEL
LIN {X 0,Y 489.983,Z 431.18,A -85,B 0,C 180,E1 23237.637,E2 23237.637} C_VEL
LIN {X 0,Y 489.982,Z 431.156,A -85,B 0,C 180,E1 23234.054,E2 23234.054} C_VEL
LIN {X 0,Y 489.98,Z 431.184,A -85,B 0,C 180,E1 23230.464,E2 23230.464} C_VEL
LIN {X 0,Y 489.971,Z 431.182,A -85,B 0,C 180,E1 23226.915,E2 23226.915} C_VEL
LIN {X 0,Y 489.982,Z 431.155,A -85,B 0,C 180,E1 23223.393,E2 23223.393} C_VEL
LIN {X 0,Y 489.997,Z 431.192,A -85,B 0,C 180,E1 23219.766,E2 23219.766} C_VEL
LIN {X 0,Y 489.971,Z 431.171,A -85,B 0,C 180,E1 23216.139,E2 23216.139} C_VEL
LIN {X 0,Y 489.952,Z 431.162,A -85,B 0,C 180,E1 23212.613,E2 23212.613} C_VEL
LIN {X 0,Y 489.977,Z 431.199,A -85,B 0,C 180,E1 23209.06,E2 23209.06} C_VEL
LIN {X 0,Y 489.996,Z 431.159,A -85,B 0,C 180,E1 23205.463,E2 23205.463} C_VEL
LIN {X 0,Y 489.953,Z 431.169,A -85,B 0,C 180,E1 23201.992,E2 23201.992} C_VEL
LIN {X 0,Y 489.94,Z 431.201,A -85,B 0,C 180,E1 23198.447,E2 23198.447} C_VEL
LIN {X 0,Y 489.973,Z 431.167,A -85,B 0,C 180,E1 23195.012,E2 23195.012} C_VEL
LIN {X 0,Y 489.956,Z 431.165,A -85,B 0,C 180,E1 23191.592,E2 23191.592} C_VEL
LIN {X 0,Y 489.926,Z 431.184,A -85,B 0,C 180,E1 23188.227,E2 23188.227} C_VEL
LIN {X 0,Y 489.949,Z 431.194,A -85,B 0,C 180,E1 23184.719,E2 23184.719} C_VEL
LIN {X 0,Y 490.003,Z 431.373,A -85,B 0,C 180,E1 23183.122,E2 23183.122} C_VEL
LIN {X 0,Y 490.349,Z 432.828,A -85,B 0,C 180,E1 23182.852,E2 23182.852} C_VEL
LIN {X 0,Y 492.259,Z 435.897,A -85,B 0,C 180,E1 23182.456,E2 23182.456} C_VEL
LIN {X 0,Y 494.485,Z 437.839,A -85,B 0,C 180,E1 23182.05,E2 23182.05} C_VEL
LIN {X 0,Y 497.003,Z 441.635,A -85,B 0,C 180,E1 23181.562,E2 23181.562} C_VEL
LIN {X 0,Y 499.011,Z 443.716,A -85,B 0,C 180,E1 23181.203,E2 23181.203} C_VEL
LIN {X 0,Y 502.257,Z 448,A -85,B 0,C 180,E1 23180.612,E2 23180.612} C_VEL
LIN {X 0,Y 508.072,Z 455.579,A -85,B 0,C 180,E1 23179.593,E2 23179.593} C_VEL
LIN {X 0,Y 515.502,Z 465.476,A -85,B 0,C 180,E1 23178.35,E2 23178.35} C_VEL
LIN {X 0,Y 528.824,Z 484.102,A -85,B 0,C 180,E1 23176.265,E2 23176.265} C_VEL
LIN {X 0,Y 542.062,Z 504.22,A -85,B 0,C 180,E1 23174.34,E2 23174.34} C_VEL
LIN {X 0,Y 546.005,Z 510.773,A -85,B 0,C 180,E1 23173.786,E2 23173.786} C_VEL
LIN {X 0,Y 537.517,Z 754.629,A -85,B 0,C 180,E1 23170.244,E2 23170.244} C_VEL
LIN {X 0,Y 535.412,Z 812.081,A -85,B 0,C 180,E1 23169.385,E2 23169.385} C_VEL
LIN {X 0,Y 533.676,Z 836.381,A -85,B 0,C 180,E1 23168.847,E2 23168.847} C_VEL
LIN {X 0,Y 531.63,Z 858.123,A -85,B 0,C 180,E1 23168.213,E2 23168.213} C_VEL
LIN {X 0,Y 528.802,Z 882.417,A -85,B 0,C 180,E1 23167.303,E2 23167.303} C_VEL
LIN {X 0,Y 525.923,Z 903.239,A -85,B 0,C 180,E1 23166.344,E2 23166.344} C_VEL
LIN {X 0,Y 522.253,Z 926.522,A -85,B 0,C 180,E1 23165.056,E2 23165.056} C_VEL
LIN {X 0,Y 518.847,Z 945.92,A -85,B 0,C 180,E1 23163.778,E2 23163.778} C_VEL
LIN {X 0,Y 514.962,Z 966.51,A -85,B 0,C 180,E1 23162.208,E2 23162.208} C_VEL
LIN {X 0,Y 511.785,Z 982.184,A -85,B 0,C 180,E1 23160.821,E2 23160.821} C_VEL
LIN {X 0,Y 509.675,Z 988.22,A -85,B 0,C 180,E1 23160.312,E2 23160.312} C_VEL
LIN {X 0,Y 500.963,Z 1004.038,A -85,B 0,C 180,E1 23159.057,E2 23159.057} C_VEL
LIN {X 0,Y 499.238,Z 1008.711,A -85,B 0,C 180,E1 23158.556,E2 23158.556} C_VEL
LIN {X 0,Y 495.733,Z 1024.391,A -85,B 0,C 180,E1 23156.601,E2 23156.601} C_VEL
LIN {X 0,Y 492.09,Z 1040.765,A -85,B 0,C 180,E1 23154.233,E2 23154.233} C_VEL
LIN {X 0,Y 489.304,Z 1053.666,A -85,B 0,C 180,E1 23152.086,E2 23152.086} C_VEL
LIN {X 0,Y 486.385,Z 1067.936,A -85,B 0,C 180,E1 23149.328,E2 23149.328} C_VEL
LIN {X 0,Y 484.379,Z 1078.551,A -85,B 0,C 180,E1 23146.922,E2 23146.922} C_VEL
LIN {X 0,Y 482.599,Z 1089.365,A -85,B 0,C 180,E1 23144.029,E2 23144.029} C_VEL
LIN {X 0,Y 481.508,Z 1097.184,A -85,B 0,C 180,E1 23141.499,E2 23141.499} C_VEL
LIN {X 0,Y 480.695,Z 1104.539,A -85,B 0,C 180,E1 23138.613,E2 23138.613} C_VEL
LIN {X 0,Y 480.257,Z 1109.659,A -85,B 0,C 180,E1 23135.975,E2 23135.975} C_VEL
LIN {X 0,Y 480.049,Z 1113.354,A -85,B 0,C 180,E1 23133.463,E2 23133.463} C_VEL
LIN {X 0,Y 479.98,Z 1116.192,A -85,B 0,C 180,E1 23130.477,E2 23130.477} C_VEL
LIN {X 0,Y 479.955,Z 1117.242,A -85,B 0,C 180,E1 23127.97,E2 23127.97} C_VEL
LIN {X 0,Y 479.943,Z 1117.175,A -85,B 0,C 180,E1 23125.459,E2 23125.459} C_VEL
LIN {X 0,Y 479.981,Z 1115.641,A -85,B 0,C 180,E1 23122.57,E2 23122.57} C_VEL
LIN {X 0,Y 480.084,Z 1112.978,A -85,B 0,C 180,E1 23120.045,E2 23120.045} C_VEL
LIN {X 0,Y 480.327,Z 1109.133,A -85,B 0,C 180,E1 23117.497,E2 23117.497} C_VEL
LIN {X 0,Y 480.922,Z 1102.837,A -85,B 0,C 180,E1 23114.442,E2 23114.442} C_VEL
LIN {X 0,Y 481.739,Z 1096.231,A -85,B 0,C 180,E1 23111.92,E2 23111.92} C_VEL
LIN {X 0,Y 483.157,Z 1087.013,A -85,B 0,C 180,E1 23109.021,E2 23109.021} C_VEL
LIN {X 0,Y 484.928,Z 1077.008,A -85,B 0,C 180,E1 23106.421,E2 23106.421} C_VEL
LIN {X 0,Y 487.415,Z 1064.772,A -85,B 0,C 180,E1 23103.698,E2 23103.698} C_VEL
LIN {X 0,Y 490.273,Z 1051.65,A -85,B 0,C 180,E1 23101.229,E2 23101.229} C_VEL
LIN {X 0,Y 493.763,Z 1036.637,A -85,B 0,C 180,E1 23098.774,E2 23098.774} C_VEL
LIN {X 0,Y 497.435,Z 1020.928,A -85,B 0,C 180,E1 23096.58,E2 23096.58} C_VEL
LIN {X 0,Y 501.537,Z 1003.655,A -85,B 0,C 180,E1 23094.468,E2 23094.468} C_VEL
LIN {X 0,Y 505.676,Z 985.528,A -85,B 0,C 180,E1 23092.579,E2 23092.579} C_VEL
LIN {X 0,Y 509.949,Z 966.493,A -85,B 0,C 180,E1 23090.849,E2 23090.849} C_VEL
LIN {X 0,Y 514.089,Z 946.393,A -85,B 0,C 180,E1 23089.297,E2 23089.297} C_VEL
LIN {X 0,Y 517.711,Z 927.543,A -85,B 0,C 180,E1 23088.037,E2 23088.037} C_VEL
LIN {X 0,Y 521.693,Z 904.621,A -85,B 0,C 180,E1 23086.746,E2 23086.746} C_VEL
LIN {X 0,Y 524.804,Z 884.15,A -85,B 0,C 180,E1 23085.787,E2 23085.787} C_VEL
LIN {X 0,Y 527.874,Z 860.574,A -85,B 0,C 180,E1 23084.878,E2 23084.878} C_VEL
LIN {X 0,Y 530.208,Z 837.974,A -85,B 0,C 180,E1 23084.204,E2 23084.204} C_VEL
LIN {X 0,Y 532.145,Z 813.866,A -85,B 0,C 180,E1 23083.656,E2 23083.656} C_VEL
LIN {X 0,Y 534.248,Z 763.229,A -85,B 0,C 180,E1 23082.879,E2 23082.879} C_VEL
LIN {X 0,Y 543.794,Z 519.46,A -85,B 0,C 180,E1 23079.282,E2 23079.282} C_VEL
LIN {X 0,Y 543.784,Z 515.553,A -85,B 0,C 180,E1 23079.204,E2 23079.204} C_VEL
LIN {X 0,Y 532.263,Z 498.117,A -85,B 0,C 180,E1 23077.374,E2 23077.374} C_VEL
LIN {X 0,Y 520.34,Z 481.337,A -85,B 0,C 180,E1 23075.339,E2 23075.339} C_VEL
LIN {X 0,Y 512.283,Z 470.671,A -85,B 0,C 180,E1 23073.866,E2 23073.866} C_VEL
LIN {X 0,Y 505.014,Z 461.257,A -85,B 0,C 180,E1 23072.45,E2 23072.45} C_VEL
LIN {X 0,Y 500.257,Z 455.402,A -85,B 0,C 180,E1 23071.478,E2 23071.478} C_VEL
LIN {X 0,Y 496.83,Z 450.904,A -85,B 0,C 180,E1 23070.743,E2 23070.743} C_VEL
LIN {X 0,Y 492.845,Z 446.313,A -85,B 0,C 180,E1 23069.873,E2 23069.873} C_VEL
LIN {X 0,Y 491.496,Z 444.417,A -85,B 0,C 180,E1 23069.56,E2 23069.56} C_VEL
LIN {X 0,Y 488.496,Z 441.484,A -85,B 0,C 180,E1 23068.886,E2 23068.886} C_VEL
LIN {X 0,Y 486.807,Z 438.536,A -85,B 0,C 180,E1 23068.459,E2 23068.459} C_VEL
LIN {X 0,Y 483.626,Z 436.065,A -85,B 0,C 180,E1 23067.722,E2 23067.722} C_VEL
LIN {X 0,Y 482.173,Z 433.058,A -85,B 0,C 180,E1 23067.277,E2 23067.277} C_VEL
LIN {X 0,Y 482.047,Z 432.197,A -85,B 0,C 180,E1 23066.882,E2 23066.882} C_VEL
LIN {X 0,Y 482.004,Z 432.166,A -85,B 0,C 180,E1 23063.342,E2 23063.342} C_VEL
LIN {X 0,Y 482,Z 432.161,A -85,B 0,C 180,E1 23059.764,E2 23059.764} C_VEL
LIN {X 0,Y 482.033,Z 432.154,A -85,B 0,C 180,E1 23056.262,E2 23056.262} C_VEL
LIN {X 0,Y 482.044,Z 432.17,A -85,B 0,C 180,E1 23052.824,E2 23052.824} C_VEL
LIN {X 0,Y 482.016,Z 432.188,A -85,B 0,C 180,E1 23049.312,E2 23049.312} C_VEL
LIN {X 0,Y 482.02,Z 432.163,A -85,B 0,C 180,E1 23045.714,E2 23045.714} C_VEL
LIN {X 0,Y 482.045,Z 432.146,A -85,B 0,C 180,E1 23042.14,E2 23042.14} C_VEL
LIN {X 0,Y 482.051,Z 432.161,A -85,B 0,C 180,E1 23038.574,E2 23038.574} C_VEL
LIN {X 0,Y 482.04,Z 432.182,A -85,B 0,C 180,E1 23034.883,E2 23034.883} C_VEL
LIN {X 0,Y 482.031,Z 432.162,A -85,B 0,C 180,E1 23031.29,E2 23031.29} C_VEL
LIN {X 0,Y 482.045,Z 432.149,A -85,B 0,C 180,E1 23027.664,E2 23027.664} C_VEL
LIN {X 0,Y 482.042,Z 432.16,A -85,B 0,C 180,E1 23024.109,E2 23024.109} C_VEL
LIN {X 0,Y 482.048,Z 432.177,A -85,B 0,C 180,E1 23020.491,E2 23020.491} C_VEL
LIN {X 0,Y 482.045,Z 432.15,A -85,B 0,C 180,E1 23016.919,E2 23016.919} C_VEL
LIN {X 0,Y 482.047,Z 432.137,A -85,B 0,C 180,E1 23013.382,E2 23013.382} C_VEL
LIN {X 0,Y 482.096,Z 432.493,A -85,B 0,C 180,E1 23011.533,E2 23011.533} C_VEL
LIN {X 0,Y 483.664,Z 436.084,A -85,B 0,C 180,E1 23010.526,E2 23010.526} C_VEL
LIN {X 0,Y 484.761,Z 438.285,A -85,B 0,C 180,E1 23009.919,E2 23009.919} C_VEL
LIN {X 0,Y 486.983,Z 442.186,A -85,B 0,C 180,E1 23008.893,E2 23008.893} C_VEL
LIN {X 0,Y 490.302,Z 446.695,A -85,B 0,C 180,E1 23008.082,E2 23008.082} C_VEL
LIN {X 0,Y 499.344,Z 458.652,A -85,B 0,C 180,E1 23006.07,E2 23006.07} C_VEL
LIN {X 0,Y 508.744,Z 471.54,A -85,B 0,C 180,E1 23004.148,E2 23004.148} C_VEL
LIN {X 0,Y 521.1,Z 489.762,A -85,B 0,C 180,E1 23001.823,E2 23001.823} C_VEL
LIN {X 0,Y 533.048,Z 508.691,A -85,B 0,C 180,E1 22999.763,E2 22999.763} C_VEL
LIN {X 0,Y 543.755,Z 527.135,A -85,B 0,C 180,E1 22998.036,E2 22998.036} C_VEL
LIN {X 0,Y 535.243,Z 746.417,A -85,B 0,C 180,E1 22994.79,E2 22994.79} C_VEL
LIN {X 0,Y 531.676,Z 837.978,A -85,B 0,C 180,E1 22993.418,E2 22993.418} C_VEL
LIN {X 0,Y 529.588,Z 863.695,A -85,B 0,C 180,E1 22992.876,E2 22992.876} C_VEL
LIN {X 0,Y 527.358,Z 884.014,A -85,B 0,C 180,E1 22992.307,E2 22992.307} C_VEL
LIN {X 0,Y 524.372,Z 906.979,A -85,B 0,C 180,E1 22991.496,E2 22991.496} C_VEL
LIN {X 0,Y 521.032,Z 928.527,A -85,B 0,C 180,E1 22990.54,E2 22990.54} C_VEL
LIN {X 0,Y 517.532,Z 948.922,A -85,B 0,C 180,E1 22989.468,E2 22989.468} C_VEL
LIN {X 0,Y 513.287,Z 971.243,A -85,B 0,C 180,E1 22988.065,E2 22988.065} C_VEL
LIN {X 0,Y 509.458,Z 989.984,A -85,B 0,C 180,E1 22986.684,E2 22986.684} C_VEL
LIN {X 0,Y 504.852,Z 1011.394,A -85,B 0,C 180,E1 22984.848,E2 22984.848} C_VEL
LIN {X 0,Y 501.053,Z 1028.423,A -85,B 0,C 180,E1 22983.147,E2 22983.147} C_VEL
LIN {X 0,Y 497.091,Z 1046.189,A -85,B 0,C 180,E1 22981.128,E2 22981.128} C_VEL
LIN {X 0,Y 493.391,Z 1062.485,A -85,B 0,C 180,E1 22978.97,E2 22978.97} C_VEL
LIN {X 0,Y 490.11,Z 1077.765,A -85,B 0,C 180,E1 22976.669,E2 22976.669} C_VEL
LIN {X 0,Y 487.103,Z 1092.299,A -85,B 0,C 180,E1 22974.11,E2 22974.11} C_VEL
LIN {X 0,Y 484.861,Z 1104.408,A -85,B 0,C 180,E1 22971.663,E2 22971.663} C_VEL
LIN {X 0,Y 482.911,Z 1116.252,A -85,B 0,C 180,E1 22968.845,E2 22968.845} C_VEL
LIN {X 0,Y 481.652,Z 1125.43,A -85,B 0,C 180,E1 22966.275,E2 22966.275} C_VEL
LIN {X 0,Y 480.695,Z 1134.396,A -85,B 0,C 180,E1 22963.223,E2 22963.223} C_VEL
LIN {X 0,Y 480.239,Z 1140.421,A -85,B 0,C 180,E1 22960.661,E2 22960.661} C_VEL
LIN {X 0,Y 479.988,Z 1145.673,A -85,B 0,C 180,E1 22957.782,E2 22957.782} C_VEL
LIN {X 0,Y 479.93,Z 1148.945,A -85,B 0,C 180,E1 22955.14,E2 22955.14} C_VEL
LIN {X 0,Y 479.928,Z 1150.717,A -85,B 0,C 180,E1 22952.866,E2 22952.866} C_VEL
LIN {X 0,Y 479.945,Z 1151.563,A -85,B 0,C 180,E1 22950.239,E2 22950.239} C_VEL
LIN {X 0,Y 479.933,Z 1150.827,A -85,B 0,C 180,E1 22947.373,E2 22947.373} C_VEL
